(* CODESYS project CtaSysIO_1.0.0.1.library
   DocFormat: reStructuredText
   DefaultNamespace: CtaSysIO
   Version: 1.0.0.1
   Placeholder: CtaSysIO
   Company: CTA
   Description: Io System Library der CTA
   CompiledLibraryCompatibilityVersion: CODESYS V3.5 SP16 Patch 3
   LanguageModelAttribute: qualified-access-only
   Title: CtaSysIO
   Author: SIS

Project tree, tasks and I/O mapping:
  libraries: WagoSysDynamicIoMapping, 1.0.4.0 (WAGO); Standard, 3.5.18.0 (System); VisuDialogs, * (System); CtaSysConfig, 1.0.0.2 (CTA); CtaVisSymbols, 1.0.0.0 (CTA); VisuSymbols, 4.5.0.0 (System); CtaAppReport, 1.0.0.2 (CTA); CtaAppBmk, 1.0.0.0 (CTA); CtaAppInfluxLog, 1.0.0.1 (CTA); SysCom, 3.5.17.0 (System); CtaSysIO, 1.0.0.1 (CTA); CtaVisHelp, 1.0.0.0 (CTA); WagoSysVisuBACnet, 2.0.0.0 (WAGO); WagoVisuIcons, 1.1.0.5 (WAGO); WagoVisuIconsMaterialDesign, 1.0.0.0 (WAGO)
  40 Visualizations/
    AI/
      visualisation SimAI_Temp
      visualisation SimAI
      visualisation SimAI_Temp_Querry
    AO/
      visualisation SimAO_Temp
      visualisation SimAO
      visualisation SimAO_Temp_Querry
    DI/
      visualisation SimDI
      visualisation SimDI_Temp
      visualisation SimDI_Temp_Querry
    DO/
      visualisation SimDO_Temp
      visualisation SimDO
      visualisation SimDO_Temp_Querry
    Simulation/
      visualisation Simulation
      visualisation ModulInfos
      visualisation SimulationInfos
      visualisation DIA_IO_CONFIG
    Parameter/
      visualisation VIS_IO_PARAMETER_BASE
      Parameter_AI/
        visualisation VIS_PARAMETER_AI
        visualisation VIS_PARAMETER_TEMP_AI
      Parameter_DI/
        visualisation VIS_PARAMETER_DI
        visualisation VIS_PARAMETER_TEMP_DI
      Parameter_AO/
        visualisation VIS_PARAMETER_AO
        visualisation VIS_PARAMETER_TEMP_AO
      Parameter_DO/
        visualisation VIS_PARAMETER_DO
        visualisation VIS_PARAMETER_TEMP_DO
    PFC VISU/
      visualisation IO_ManagerBusInfo
      visualisation PFC_SLOT
      visualisation IO_Manager_Base
      visualisation IO_Manager_Sync
      visualisation IO_Manager_View
  30 Program Organization Units/
    fb/
      function block fbIO_Manager_Alt [ST]: proCycleStartDelayDone, metRequestIO_ITF, proAyIOs, proMaxIO, proErrNotEnoughIOs, proIoInitDone, proKbusErrHW, proKbusErrSW, proNeededMemSize, metRequestCOM_ITF, metModulConfigCheck
      HilfsFbs/
        function block fbIO [ST]: proSimVisu, proSlot, proChannelAdress, proPhysikalValueVisu, proOK, proKbusOk, proChannel, metCyclicKbus, proModuleType, proOkVisu, metConfig, P_scfbIO_fbxSimulationLock, P_scfbIO_Simulation, proIsHand, proAyPos, metTrendLog, proLogName, proIsBOOL_IO, proIoSim
        function block fbAI [ST]: proPhysikalValueVisu, proValue, metCyclicKbus, proAlUnterlauf, proPhysicalValue, proAlUeberlauf, proThisRef_AI, P_scfbAI_fbrMin, P_scfbAI_fbrMax, P_scfbAI_fbrMinPhysical, P_scfbAI_fbstPhysicalUnit, P_scfbAI_fbrPhysicalAlarm, P_scfbAI_fbrSimulationValue, P_scfbAI_fbrCorrectionValue, P_All_Init, metConfig, metTrendLog, proLogName, proIsBOOL_IO
        function block fbDO [ST]: proPhysikalValueVisu, proValue, metCyclicKbus, metConfig, proThisRef_DO, P_scfbDO_fbxInvert, P_scfbDO_fbxSimulationValue, P_All_Init, metTrendLog, proLogName, proIsBOOL_IO
        function block fbAO [ST]: proPhysikalValueVisu, metCyclicKbus, proValue, proPhysicalValue, metConfig, proThisRef_AO, P_scfbAO_fbrMin, P_scfbAO_fbrMax, P_scfbAO_fbrMinPhysical, P_scfbAO_fbrSimulationValue, P_All_Init, metTrendLog, proLogName, proIsBOOL_IO
        function block fbDI [ST]: proPhysikalValueVisu, metCyclicKbus, proValue, metConfig, proThisRef_DI, P_scfbDI_fbxInvert, P_scfbDI_fbxSimulationValue, P_All_Init, metTrendLog, proLogName, proIsBOOL_IO
      visuhilfe/
        function block fbPfcVisuHelp [ST]: metGetSlotIos, metNotShowChannel, proScrollBar, metCalcScrollBar, metCalcSlotFromScrollBar, getSizeOfFrame
      function block fbIO_Manager [ST]: proCycleStartDelayDone, metRequestIO_ITF, proAyIOs, proMaxIO, proErrNotEnoughIOs, proIoInitDone, proKbusErrHW, proKbusErrSW, proNeededMemSize, metRequestCOM_ITF, metModulConfigCheck, proSimOn, proAllowSim
    fc/
      Modul/
        function fcModuleType [ST]
      Adresse/
        function fcSlotAdress [ST]
      Skalierungen/
        function fcScaleIN4_20mA [ST]
        function fcScalePT1000 [ST]
        function fcSimValueScaler [ST]
        function fcScaleIN0_10V [ST]
        function fcScaleOut [ST]
      ITF_Prüfung/
        function fc_ITF_Evaluation [ST]
      Terminal Visu/
        function fcGetModulImage [ST]
        function fcSetModulImageForSimAndGetChanels [ST]
      ModulCheck/
        function fcCheckModul [ST]
    program IO [ST]
  00000000-0000-0000-0000-000000000000|D:\CoDeSys\LibrariesV3\trunk\Intern\CAA\CAA Template\3.4.0.0 draft\Placeholder.xml
  00000000-0000-0000-0000-000000000000|D:\CoDeSys\LibrariesV3\trunk\Intern\CAA\CAA Template\3.2.0.3 draft\Prefix.pdf
  00000000-0000-0000-0000-000000000000|D:\CoDeSys\LibrariesV3\trunk\Intern\CAA\CAA Template\3.5.2.0 draft\Placeholder.xml
  20 Structs/
    data type scChanelAdress
    data type enModuleType
    Parameter/
      data type scAI_Para
      data type scAO_Para
      data type scDI_Para
      data type scDO_Para
  50 Images/
    image pool IO_TERMINALS
  10 Documenation/
    global variables VersionHistory
    global variables readMe
  21 Interface/
    Visu/
      interface ITF_IO_Manager_Visu: proErrNotEnoughIOs, proNeededMemSize, proIoInitDone, proKbusErrSW, proKbusErrHW, proMaxIO, proAyIOs, proSimOn, proAllowSim
    IO/
      interface ITF_AI: proAlUnterlauf, proValue, proPhysicalValue, proAlUeberlauf, proThisRef_AI, P_scfbAI_fbrCorrectionValue, P_scfbAI_fbrMax, P_scfbAI_fbrMin, P_scfbAI_fbrMinPhysical, P_scfbAI_fbrPhysicalAlarm, P_scfbAI_fbrSimulationValue, P_scfbAI_fbstPhysicalUnit, P_All_Init
      interface ITF_AO: proPhysicalValue, proValue, proThisRef_AO, P_scfbAO_fbrMax, P_scfbAO_fbrMin, P_scfbAO_fbrMinPhysical, P_scfbAO_fbrSimulationValue, P_All_Init
      interface ITF_DI: proValue, proThisRef_DI, P_scfbDI_fbxInvert, P_scfbDI_fbxSimulationValue, P_All_Init
      interface ITF_DO: proValue, proThisRef_DO, P_scfbDO_fbxInvert, P_scfbDO_fbxSimulationValue, P_All_Init
      interface ITF_IO: proPhysikalValueVisu, proKbusOk, proOkVisu, proModuleType, proSimVisu, proOK, proSlot, proChannel, metCyclicKbus, proChannelAdress, P_scfbIO_fbxSimulationLock, P_scfbIO_Simulation, proIsHand, proLogName, proIsBOOL_IO, proIoSim
  11 Library Parameter/
    global variables Parameter
  12 Konstanten/
    global variables GlobalKonstant
  60 Textlisten/
    text list txtModulType
    text list txtWarning
    text list txtError
    text list txtPhysicalUnit
  13 Globale Variablen/
    global variables GVL_IO
    global variables GVL_IO_TERMINALS
  text list GlobalTextList
  5ce3da45-db07-42e7-a21c-a00fff4ed8f6|S:\_Temporär_SIS\CtaCodesysLibrary\01_Library\CtaSysIO\04_Image\0750_400.bmp
  5ce3da45-db07-42e7-a21c-a00fff4ed8f6|S:\_Temporär_SIS\CtaCodesysLibrary\01_Library\CtaSysIO\04_Image\0750_432.bmp
  5ce3da45-db07-42e7-a21c-a00fff4ed8f6|S:\_Temporär_SIS\CtaCodesysLibrary\01_Library\CtaSysIO\04_Image\0750_451.bmp
  5ce3da45-db07-42e7-a21c-a00fff4ed8f6|S:\_Temporär_SIS\CtaCodesysLibrary\01_Library\CtaSysIO\04_Image\0750_455.bmp
  5ce3da45-db07-42e7-a21c-a00fff4ed8f6|S:\_Temporär_SIS\CtaCodesysLibrary\01_Library\CtaSysIO\04_Image\0750_459.bmp
  5ce3da45-db07-42e7-a21c-a00fff4ed8f6|S:\_Temporär_SIS\CtaCodesysLibrary\01_Library\CtaSysIO\04_Image\0750_466.bmp
  5ce3da45-db07-42e7-a21c-a00fff4ed8f6|S:\_Temporär_SIS\CtaCodesysLibrary\01_Library\CtaSysIO\04_Image\0750_515.bmp
  5ce3da45-db07-42e7-a21c-a00fff4ed8f6|S:\_Temporär_SIS\CtaCodesysLibrary\01_Library\CtaSysIO\04_Image\0750_597.bmp
  5ce3da45-db07-42e7-a21c-a00fff4ed8f6|S:\_Temporär_SIS\CtaCodesysLibrary\01_Library\CtaSysIO\04_Image\0750_600.bmp
  5ce3da45-db07-42e7-a21c-a00fff4ed8f6|S:\_Temporär_SIS\CtaCodesysLibrary\01_Library\CtaSysIO\04_Image\0750_652.bmp
  5ce3da45-db07-42e7-a21c-a00fff4ed8f6|S:\_Temporär_SIS\CtaCodesysLibrary\01_Library\CtaSysIO\04_Image\0750_1405.bmp
  5ce3da45-db07-42e7-a21c-a00fff4ed8f6|S:\_Temporär_SIS\CtaCodesysLibrary\01_Library\CtaSysIO\04_Image\0750_1415.bmp
  5ce3da45-db07-42e7-a21c-a00fff4ed8f6|S:\_Temporär_SIS\CtaCodesysLibrary\01_Library\CtaSysIO\04_Image\0750_1504.bmp
  5ce3da45-db07-42e7-a21c-a00fff4ed8f6|S:\_Temporär_SIS\CtaCodesysLibrary\01_Library\CtaSysIO\04_Image\0750_8212.bmp
  5ce3da45-db07-42e7-a21c-a00fff4ed8f6|S:\_Temporär_SIS\CtaCodesysLibrary\01_Library\CtaSysIO\04_Image\0750_BLANK.bmp
  5ce3da45-db07-42e7-a21c-a00fff4ed8f6|S:\_Temporär_SIS\CtaCodesysLibrary\01_Library\CtaSysIO\04_Image\0750_555.bmp
*)

// 20 Structs/scChanelAdress
TYPE scChanelAdress :
STRUCT	
	uiByteNr	: 	UINT;
	uiBitNR		:	USINT;	
END_STRUCT
END_TYPE

// 20 Structs/enModuleType
{attribute 'qualified_only'}
{attribute 'strict'}
{attribute 'to_string'}
TYPE enModuleType :
(
	Unknown 		:= 0,
	Digital_IN		:= 1,
	Digital_OUT		:= 2,	
	DC_0_10V_OUT	:= 3,
	DC_4_20mA_OUT	:= 4,
	DC_0_10V_IN		:= 5,
	DC_4_20mA_IN	:= 6,
	OHM				:= 7,
    RS485			:= 8,
	DC_0_20mA_OUT	:= 9
);
END_TYPE

// 20 Structs/Parameter/scAI_Para
TYPE scAI_Para :
	STRUCT
		xSimulationLock		:	BOOL;
		rMin				:	REAL;
		rMax				:	REAL;
		rMinPhysical		:	REAL;
		rPhysicalAlarm		:	REAL;
		rCorrectionValue	:	REAL;
		stPhysicalUnit		:	STRING(40);
	END_STRUCT
END_TYPE

// 20 Structs/Parameter/scAO_Para
TYPE scAO_Para :
	STRUCT
		xSimulationLock		:	BOOL;
		rMin				:	REAL;
		rMax				:	REAL;
		rMinPhysical		:	REAL;
	END_STRUCT
END_TYPE

// 20 Structs/Parameter/scDI_Para
TYPE scDI_Para :
	STRUCT
		xSimulationLock		:	BOOL;
		xInvert				:	BOOL;
	END_STRUCT
END_TYPE

// 20 Structs/Parameter/scDO_Para
TYPE scDO_Para :
	STRUCT
		xSimulationLock		:	BOOL;
		xInvert				:	BOOL;
	END_STRUCT
END_TYPE

// 10 Documenation/VersionHistory
(* 

.. image:: ../../Images/CTA_Logo.jpg
   :align: right
   :width: 15% 

**Vorlage**   


============ =========== =========== ============================================
**Date**     **Version** **Author**  **Change**
------------ ----------- ----------- --------------------------------------------
04.03.2021   0.0.0.0     SIS         Vorlage erstellt

============ =========== =========== ============================================


*)
VAR_GLOBAL
    stInfo : STRING:= '0.0.0.0, Vorlage, CTA';
END_VAR

// 10 Documenation/readMe
(*

**ReadMe**
 
|	**Empfehlung**
|
|	Dokumentrieren Sie die Library für eine nachhaltige Entwicklung
|     
| *Beispiel*
| 
| Dies ist die Vorlage Library der CTA. Erstellen Sie ihre Library anhand dieser Vorlage.
*)

VAR_GLOBAL
    xReadMeDone              :   BOOL;
END_VAR

// 13 Globale Variablen/GVL_IO
{attribute 'qualified_only'}
VAR_GLOBAL	
	fbIO_Manager : fbIO_Manager;
END_VAR

// 11 Library Parameter/Parameter
{attribute 'qualified_only'}
VAR_GLOBAL CONSTANT
	SPS_BMK_ID        		: STRING(20)   := 'SPS';
	MAX_NUM_OF_DI			: INT := 200;
	MAX_NUM_OF_DO			: INT := 200;
	MAX_NUM_OF_AI			: INT := 100;
	MAX_NUM_OF_AO			: INT := 100;	
	                		
	MAX_NUM_OF_IOS			: INT := MAX_NUM_OF_DI + MAX_NUM_OF_DO + MAX_NUM_OF_AI + MAX_NUM_OF_AO;
	
	MAX_NUM_OF_COMTYPES		: INT := 10;
END_VAR

// 12 Konstanten/GlobalKonstant
{attribute 'qualified_only'}
VAR_GLOBAL CONSTANT
    stWarningTextList   :   STRING  := 'CtaSysIO.txtWarning';
    stErrorTextList     :   STRING  := 'CtaSysIO.txtError';
	ayMin	: ARRAY [enModuleType.Unknown..enModuleType.DC_0_20mA_OUT] OF REAL := [3(0), 0.0, 4, 0, 4, -250, 2(0.0)];
	ayMax	: ARRAY [enModuleType.Unknown..enModuleType.DC_0_20mA_OUT] OF REAL := [0, 2(1), 10, 20, 10, 20, 850, 0.0, 20];
END_VAR

// 13 Globale Variablen/GVL_IO_TERMINALS
{attribute 'qualified_only'}
VAR_GLOBAL
	aystIoTerminalType		:	ARRAY[1..125] OF STRING;
END_VAR

// 21 Interface/IO/ITF_AI
INTERFACE ITF_AI EXTENDS ITF_IO

PROPERTY proAlUnterlauf : BOOL
GET
END_GET
END_PROPERTY

PROPERTY proValue : REAL
GET
END_GET
END_PROPERTY

PROPERTY proPhysicalValue : REAL
GET
END_GET
END_PROPERTY

PROPERTY proAlUeberlauf : BOOL
GET
END_GET
END_PROPERTY

PROPERTY proThisRef_AI : REFERENCE TO fbAI
GET
END_GET
END_PROPERTY

PROPERTY P_scfbAI_fbrCorrectionValue : CtaSysConfig.ITF_DATATYPE
GET
END_GET
END_PROPERTY

PROPERTY P_scfbAI_fbrMax : CtaSysConfig.ITF_DATATYPE
GET
END_GET
END_PROPERTY

PROPERTY P_scfbAI_fbrMin : CtaSysConfig.ITF_DATATYPE
GET
END_GET
END_PROPERTY

PROPERTY P_scfbAI_fbrMinPhysical : CtaSysConfig.ITF_DATATYPE
GET
END_GET
END_PROPERTY

PROPERTY P_scfbAI_fbrPhysicalAlarm : CtaSysConfig.ITF_DATATYPE
GET
END_GET
END_PROPERTY

PROPERTY P_scfbAI_fbrSimulationValue : CtaSysConfig.ITF_DATATYPE
GET
END_GET
END_PROPERTY

PROPERTY P_scfbAI_fbstPhysicalUnit : CtaSysConfig.ITF_DATATYPE
GET
END_GET
END_PROPERTY

PROPERTY P_All_Init : scAI_Para
SET
END_SET
END_PROPERTY

END_INTERFACE

// 21 Interface/IO/ITF_IO
INTERFACE ITF_IO EXTENDS __system.IQueryInterface

PROPERTY proPhysikalValueVisu : STRING(6)
GET
END_GET
END_PROPERTY

PROPERTY proKbusOk : BOOL
GET
END_GET
SET
END_SET
END_PROPERTY

PROPERTY proOkVisu : STRING
GET
END_GET
END_PROPERTY

PROPERTY proModuleType : enModuleType
SET
END_SET
GET
END_GET
END_PROPERTY

PROPERTY proSimVisu : STRING
GET
END_GET
END_PROPERTY

PROPERTY proOK : BOOL
GET
END_GET
END_PROPERTY

PROPERTY proSlot : USINT
SET
END_SET
GET
END_GET
END_PROPERTY

PROPERTY proChannel : UINT
GET
END_GET
SET
END_SET
END_PROPERTY

METHOD metCyclicKbus
VAR_INPUT
END_VAR
END_METHOD

PROPERTY proChannelAdress : scChanelAdress
SET
END_SET
END_PROPERTY

PROPERTY P_scfbIO_fbxSimulationLock : CtaSysConfig.ITF_DATATYPE
GET
END_GET
END_PROPERTY

PROPERTY P_scfbIO_Simulation : CtaSysConfig.ITF_DATATYPE
GET
END_GET
END_PROPERTY

PROPERTY proIsHand : BOOL
GET
END_GET
END_PROPERTY

PROPERTY proLogName : STRING(100)
GET
END_GET
END_PROPERTY

PROPERTY proIsBOOL_IO : BOOL
GET
END_GET
END_PROPERTY

PROPERTY proIoSim : BOOL
SET
END_SET
GET
END_GET
END_PROPERTY

END_INTERFACE

// 30 Program Organization Units/fb/HilfsFbs/fbAI
FUNCTION_BLOCK fbAI EXTENDS fbIO IMPLEMENTS ITF_AI

VAR
	(*Channel input*)
	wChannelIn			: 	WORD;	
	
	(*Value output*)
	rValue				: 	REAL;
	
	(*Calculation Vars*)
	rPhysicalValueSIM	:	REAL;	// Errechneter Wert V oder mA der Simulation
	rPhysicalValuePLC 	:	REAL;	// Errechneter Wert V oder mA des PGMs
	rUserScale			:	REAL;  	// Funktionsausgabe, Physikalisch oder Benutzerdefiniert skaliert	
	
	(*Alarm*)	
	xAlUeberlauf		:	BOOL;	// Alarm Überlauf
	xAlUnterlauf		:	BOOL;	// Alarm Unterlauf
	(* Trendlog *)
	fbTrendLogrValue	:	CtaAppInfluxLog.FB_LOG_NODE_REAL;		
	(*Parameter*)	
	fbrMin				:	CtaSysConfig.fbREAL;			
	fbrMax				:	CtaSysConfig.fbREAL;		
	fbrMinPhysical		:	CtaSysConfig.fbREAL;
	fbstPhysicalUnit	:	CtaSysConfig.fbSTRING40;			
	fbrPhysicalAlarm	:	CtaSysConfig.fbREAL;			
	fbrSimulationValue	:	CtaSysConfig.fbREAL;
	fbrCorrectionValue	:	CtaSysConfig.fbREAL;			
END_VAR

PROPERTY proPhysikalValueVisu : STRING(6)
GET
// Schreiben des physikalischen Wertes für Visualisierung
IF FIND(TO_STRING(proPhysicalValue),'.') <> 0 THEN
	proPhysikalValueVisu := LEFT(TO_STRING(proPhysicalValue),(FIND(TO_STRING(proPhysicalValue),'.')+1));	
ELSE
	proPhysikalValueVisu := TO_STRING(proPhysicalValue);
END_IF
END_GET
END_PROPERTY

PROPERTY proValue : REAL
GET
(*Wert mit Korrektur*)
proValue := rValue;
END_GET
END_PROPERTY

METHOD FINAL metCyclicKbus
VAR
	xTempOk	:	BOOL;
END_VAR
metConfig();

// Lesen des Wertes aus definiertem Eingang
IF usiSlot > 0 AND WagoSysDynamicIoMapping.DynIoManager.DynKbusIoManager.coModules.uiModuleCount >= usiSlot THEN
	wChannelIn := WagoSysDynamicIoMapping.DynIoManager.DynKbusIoManager.coModules.aIModules[usiSlot].GetProcessInWord(scAdressOfChanel.uiByteNr,oStatus => oStatus);
ELSE
	wChannelIn 	:= 0;
	xOK			:= FALSE;
END_IF

// Modultyp bestimmen für physikalische Einheit
CASE enTypeOfModul OF
	enModuleType.DC_0_10V_IN,enModuleType.DC_0_10V_OUT:
		fbrSimulationValue.metNewMinMax(0,10); 
	enModuleType.DC_0_20mA_OUT:
		fbrSimulationValue.metNewMinMax(0,20); 
	enModuleType.DC_4_20mA_IN,enModuleType.DC_4_20mA_OUT:
		fbrSimulationValue.metNewMinMax(4,20);
	enModuleType.OHM:
		fbrSimulationValue.metNewMinMax(-2000,8500);
END_CASE	

// Signalausgabe an PGM, bei aktiver Simulation = Simulationswert
IF NOT fbxSimulation.xValue OR fbxSimulationLock.xValue THEN
      // Skalierung 0-10 V
	IF enTypeOfModul = enModuleType.DC_0_10V_IN THEN
		
		rUserScale := fcScaleIN0_10V(	wChanelInput 	:= 	wChannelIn,
										rMin 			:= 	fbrMin.rValue,
										rMax 			:= 	fbrMax.rValue,
										rMinPysical 	:=	fbrMinPhysical.rValue,
										rPysicalAlarm	:=	fbrPhysicalAlarm.rValue,									
										xOk				:= 	xOK,
										rV 				 => rPhysicalValuePLC,
										xAlUeberlauf 	 => xAlUeberlauf,
										xAlUnterlauf 	 => xAlUnterlauf);
										
	// Skalierung 4-20 mA	
	ELSIF enTypeOfModul = enModuleType.DC_4_20mA_IN THEN
	
		rUserScale := fcScaleIN4_20mA(	wChanelInput 	:= 	wChannelIn,
										rMin			:= 	fbrMin.rValue,
										rMax 			:= 	fbrMax.rValue,
										rmA 			 => rPhysicalValuePLC,
										xOK 			 => xOK,
										xAlUeberlauf 	 => xAlUeberlauf,
										xAlUnterlauf 	 => xAlUnterlauf);	

	// Skalierung ohm	
	ELSIF enTypeOfModul = enModuleType.ohm THEN
		
		rUserScale := fcScalePT1000(	wChanelInput	:=	wChannelIn,
										xOK 			 => xOK,
										xAlUeberlauf 	 => xAlUeberlauf,
										xAlUnterlauf 	 => xAlUnterlauf);
										
		rPhysicalValuePLC := rUserScale;

	END_IF
	
	// Übergabe des skalierten Eingangssignals
	rValue						:= rUserScale  + fbrCorrectionValue.rValue;
	fbrSimulationValue.metNewValueNoSave(proPhysicalValue);      
ELSE
	IF enTypeOfModul = enModuleType.ohm THEN
		rValue              := fbrSimulationValue.rValue;
		rPhysicalValueSIM   := fbrSimulationValue.rValue;    
	ELSE	
		// Skalierung des Simulationswertes
		rValue := fcSimValueScaler(	rSimulationValue 	:=	fbrSimulationValue.rValue,
									enIOModulType		:=	enTypeOfModul,
									rMin 				:= 	fbrMin.rValue,
									rMinPysical			:=	fbrMinPhysical.rValue,
									rMax				:=	fbrMax.rValue,
									rPysicalAlarm 		:=	fbrPhysicalAlarm.rValue,
									xOk 				:= 	xOK,
									xAlUnterlauf 		 => xAlUnterlauf);
		rPhysicalValueSIM := fbrSimulationValue.rValue;
	END_IF
END_IF

(* TREND *)
metTrendLog();
END_METHOD

PROPERTY proAlUnterlauf : BOOL
GET
proAlUnterlauf := xAlUnterlauf;
END_GET
END_PROPERTY

PROPERTY proPhysicalValue : REAL
GET
// Ausgabe Simulationswert bei aktiver Simulation
IF fbxSimulation.proValue THEN
	proPhysicalValue := rPhysicalValueSIM;
ELSE
	proPhysicalValue := rPhysicalValuePLC;
END_IF
END_GET
END_PROPERTY

PROPERTY proAlUeberlauf : BOOL
GET
proAlUeberlauf := xAlUeberlauf;
END_GET
END_PROPERTY

PROPERTY proThisRef_AI : REFERENCE TO fbAI
GET
proThisRef_AI REF= THIS^;
END_GET
END_PROPERTY

PROPERTY P_scfbAI_fbrMin : CtaSysConfig.ITF_DATATYPE
GET
P_scfbAI_fbrMin := fbrMin;
END_GET
END_PROPERTY

PROPERTY P_scfbAI_fbrMax : CtaSysConfig.ITF_DATATYPE
GET
P_scfbAI_fbrMax := fbrMax;
END_GET
END_PROPERTY

PROPERTY P_scfbAI_fbrMinPhysical : CtaSysConfig.ITF_DATATYPE
GET
P_scfbAI_fbrMinPhysical:= fbrMinPhysical;
END_GET
END_PROPERTY

PROPERTY P_scfbAI_fbstPhysicalUnit : CtaSysConfig.ITF_DATATYPE
GET
P_scfbAI_fbstPhysicalUnit := fbstPhysicalUnit;
END_GET
END_PROPERTY

PROPERTY P_scfbAI_fbrPhysicalAlarm : CtaSysConfig.ITF_DATATYPE
GET
P_scfbAI_fbrPhysicalAlarm := fbrPhysicalAlarm;
END_GET
END_PROPERTY

PROPERTY P_scfbAI_fbrSimulationValue : CtaSysConfig.ITF_DATATYPE
GET
P_scfbAI_fbrSimulationValue := fbrSimulationValue;
END_GET
END_PROPERTY

PROPERTY P_scfbAI_fbrCorrectionValue : CtaSysConfig.ITF_DATATYPE
GET
P_scfbAI_fbrCorrectionValue := fbrCorrectionValue;
END_GET
END_PROPERTY

PROPERTY P_All_Init : scAI_Para
SET
fbxSimulationLock._WertInit 	:= P_All_Init.xSimulationLock;
fbrMin._WertInit				:= P_All_Init.rMin;
fbrMax._WertInit				:= P_All_Init.rMax;
fbrMinPhysical._WertInit		:= P_All_Init.rMinPhysical;
fbrPhysicalAlarm._WertInit		:= P_All_Init.rPhysicalAlarm;
fbrCorrectionValue._WertInit	:= P_All_Init.rCorrectionValue;
fbstPhysicalUnit._WertInit		:= P_All_Init.stPhysicalUnit;
END_SET
END_PROPERTY

METHOD metConfig
VAR_INPUT
END_VAR
fbConfigFile();

fbxSimulation 					(_usiParaNr := 1, itfConfigFb := fbConfigFile);
fbxSimulationLock				(_usiParaNr := 2, itfConfigFb := fbConfigFile);
fbrMin							(_usiParaNr := 3, itfConfigFb := fbConfigFile);
fbrMax							(_usiParaNr := 4, itfConfigFb := fbConfigFile);
fbrMinPhysical					(_usiParaNr := 5, itfConfigFb := fbConfigFile);
fbrPhysicalAlarm				(_usiParaNr := 6, itfConfigFb := fbConfigFile);
fbrSimulationValue				(_usiParaNr := 7, itfConfigFb := fbConfigFile);
fbrCorrectionValue				(_usiParaNr := 8, itfConfigFb := fbConfigFile);
fbstPhysicalUnit				(_usiParaNr := 9, itfConfigFb := fbConfigFile);
END_METHOD

METHOD metTrendLog
IF NOT fbTrendLogrValue.ENABLE THEN
	fbTrendLogrValue.ENABLE	 := TRUE;
	fbTrendLogrValue.KEY	 := CONCAT('SLOT_',CONCAT(TO_STRING(usiSlot),CONCAT('_AI_',TO_STRING(uiChanel))));
END_IF;
fbTrendLogrValue.SET_VALUE	 := SEL(proIsHand,rPhysicalValuePLC,rPhysicalValueSIM);
END_METHOD

PROPERTY proLogName : STRING(100)
GET
proLogName := CONCAT('SLOT_',CONCAT(TO_STRING(usiSlot),CONCAT('_AI_',TO_STRING(uiChanel))));
END_GET
END_PROPERTY

PROPERTY proIsBOOL_IO : BOOL
GET
proIsBOOL_IO := FALSE;
END_GET
END_PROPERTY

END_FUNCTION_BLOCK

// 30 Program Organization Units/fb/HilfsFbs/fbIO
FUNCTION_BLOCK fbIO IMPLEMENTS ITF_IO
VAR_INPUT
END_VAR
VAR_OUTPUT
END_VAR
VAR	
	iAyPos				:	INT;
	xOK					: 	BOOL;
	xKbusOk				:	BOOL;
	xIoSim				:	BOOL;
	usiSlot				:	USINT;
	uiChanel			:	UINT;
	enTypeOfModul		:	enModuleType;
	scAdressOfChanel	: 	scChanelAdress;
	oStatus				: 	WagoSysErrorBase.FbResult;	
	
	(*Parameter*)
	fbConfigFile		: 	CtaSysConfig.fbConfigFile;

	fbxSimulation		:	CtaSysConfig.fbBOOL;
	fbxSimulationLock	:	CtaSysConfig.fbBOOL;	

END_VAR

PROPERTY proSimVisu : STRING
GET
// Simbolausgabe für Visu bei aktiver Simulations- Sperre
IF fbxSimulationLock.proValue THEN	
	proSimVisu := 'CtaVisSymbols.ImagePool.lock_closed_black';	
ELSE	
	IF fbxSimulation.proValue THEN
		proSimVisu := 'CtaVisSymbols.ImagePool.front_hand_Yellow';
	ELSE
		proSimVisu := '';
	END_IF	
END_IF
END_GET
END_PROPERTY

PROPERTY proSlot : USINT
SET
usislot := proSlot;
END_SET
GET
proSlot := usislot;
END_GET
END_PROPERTY

PROPERTY proChannelAdress : scChanelAdress
SET
scAdressOfChanel := proChannelAdress;
END_SET
END_PROPERTY

PROPERTY proPhysikalValueVisu : STRING(6)
GET
END_GET
SET
END_SET
END_PROPERTY

PROPERTY proOK : BOOL
GET
// Setzen des Modul OKs 
IF xOK AND xKbusOk THEN
	proOK := TRUE;
ELSIF xIoSim THEN
	proOK := TRUE;
ELSE
	proOK := FALSE;
END_IF
END_GET
END_PROPERTY

PROPERTY proKbusOk : BOOL
GET
 proKbusOk := xKbusOk;
END_GET
SET
xKbusOk := proKbusOk;
END_SET
END_PROPERTY

PROPERTY proChannel : UINT
SET
uiChanel := proChannel;
END_SET
GET
proChannel := uiChanel;
END_GET
END_PROPERTY

METHOD metCyclicKbus
END_METHOD

PROPERTY proModuleType : enModuleType
GET
proModuleType := enTypeOfModul;
END_GET
SET
enTypeOfModul := proModuleType;
END_SET
END_PROPERTY

PROPERTY proOkVisu : STRING
GET
// Definition des anzuzeigenden Bildes für Visu
IF xOK AND xKbusOk THEN
	proOkVisu := 'CtaVisSymbols.ImagePool.check_green';
ELSIF xIoSim THEN
	proOkVisu := 'CtaVisSymbols.ImagePool.front_hand_Yellow';
ELSE
	proOkVisu := 'CtaVisSymbols.ImagePool.CtaError';
END_IF
END_GET
END_PROPERTY

METHOD metConfig
VAR_INPUT
END_VAR
fbConfigFile();

fbxSimulation 					(_usiParaNr := 1, itfConfigFb := fbConfigFile,);
fbxSimulationLock				(_usiParaNr := 2, itfConfigFb := fbConfigFile,);
END_METHOD

PROPERTY P_scfbIO_fbxSimulationLock : CtaSysConfig.ITF_DATATYPE
GET
P_scfbIO_fbxSimulationLock := fbxSimulationLock;
END_GET
END_PROPERTY

PROPERTY P_scfbIO_Simulation : CtaSysConfig.ITF_DATATYPE
GET
P_scfbIO_Simulation := fbxSimulation;
END_GET
END_PROPERTY

PROPERTY proIsHand : BOOL
GET
proIsHand := NOT fbxSimulationLock.xValue AND fbxSimulation.xValue;
END_GET
END_PROPERTY

PROPERTY proAyPos : UINT
SET
iAyPos := TO_INT(proAyPos);
END_SET
GET
proAyPos := TO_UINT(iAyPos);
END_GET
END_PROPERTY

METHOD metTrendLog
END_METHOD

PROPERTY proLogName : STRING(100)
GET
proLogName := '';
END_GET
END_PROPERTY

PROPERTY proIsBOOL_IO : BOOL
GET
proIsBOOL_IO := FALSE;
END_GET
END_PROPERTY

PROPERTY proIoSim : BOOL
SET
xIoSim := proIoSim;
END_SET
GET
proiosim := xIoSim;
END_GET
END_PROPERTY

END_FUNCTION_BLOCK

// 30 Program Organization Units/fc/Skalierungen/fcScaleIN0_10V
FUNCTION fcScaleIN0_10V : Real
VAR_INPUT
	wChanelInput	: WORD;
	
	// Values for scaling
	rMin			:	REAL;
	rMinPysical		:	REAL;
	rMax			:	REAL;	
	rPysicalAlarm	:	REAL;	
END_VAR
VAR
	iChanelInput	: INT;
END_VAR
VAR_OUTPUT
	rV				: REAL;
	xAlUeberlauf	: BOOL;
	xAlUnterlauf	: BOOL;
END_VAR
VAR_IN_OUT
	xOk				: 	BOOL;
END_VAR

IF wChanelInput.0 = FALSE AND wChanelInput.1 = FALSE THEN
	// Für 12Bit Messwertausgabe die 3 Status Bit weglassen. Bit 16 kann vernachläsigt werden, da es immer 0 ist.
	iChanelInput 			:= WORD_TO_INT(SHR(wChanelInput,3)); 			// Prozesswert des AD Wandlers in INT										
	rV	   					:= INT_TO_REAL(iChanelInput) /(4095.0/10.0);	// Skalierung des Messwertes auf 0-10V
	// Prüfen ob die Skalierung machbar ist
	IF rMax - rMin <> 0 THEN	
		// Skalieren des Messwertes
		fcScaleIN0_10V		:= (INT_TO_REAL(iChanelInput)-(rMinPysical*4095/10)) * ((  rMax - rMin)/(4095.0-(rMinPysical*4095/10))) + rMin;  
	ELSE
		fcScaleIN0_10V		:= rV;	
	END_IF;
	// Schaltung: Messwert in Range
    IF rV >= rMinPysical THEN
        xOK             	:= TRUE;
	ELSIF rV < rMinPysical AND rV > (rMinPysical-((rMinPysical - rPysicalAlarm)/3)) THEN
		fcScaleIN0_10V  	:= rMin;
	ELSIF rV <= (rMinPysical-((rMinPysical - rPysicalAlarm)/3)) THEN
		xOK             	:= FALSE;    
        fcScaleIN0_10V  	:= rMin;
    END_IF;
	    
	// Störung: Sensorleitung ist Unterbrochen		
	IF rV < rPysicalAlarm THEN
        fcScaleIN0_10V   	:= 0; 	
        xAlUnterlauf     	:= TRUE;
        xOK              	:= FALSE;
	END_IF;
// Störung: Sensorleitung ist Unterbrochen	
ELSIF wChanelInput.0 = TRUE	AND wChanelInput.1 = TRUE THEN
	xAlUnterlauf			:= TRUE;
    fcScaleIN0_10V			:= -3.402823E+38;
	xOK						:= FALSE;
// Störung: Sensorleitung hat Überlauf	
ELSIF wChanelInput.0 = TRUE AND wChanelInput.1 = FALSE THEN
	xAlUeberlauf            := TRUE;
   	fcScaleIN0_10V          := 3.402823E+38;
	xOK						:= FALSE;
END_IF

END_FUNCTION

// 30 Program Organization Units/fc/Skalierungen/fcScaleIN4_20mA
FUNCTION fcScaleIN4_20mA : REAL
VAR_INPUT
	wChanelInput	: WORD;
	rMin        	: REAL;
    rMax        	: REAL;  
END_VAR	
VAR
	iChanelInput	: INT;	
END_VAR
VAR_OUTPUT
	rmA				: REAL;
	xOK				: BOOL;
	xAlUeberlauf	: BOOL;
	xAlUnterlauf	: BOOL;
END_VAR

//  Prüfen der Error Bit 0 & Bit 1 
IF wChanelInput.0 = FALSE AND wChanelInput.1 = FALSE THEN
	// Für 12Bit Messwertausgabe die 3 Status Bit weglassen. Bit 16 kann vernachläsigt werden, da es immer 0 ist.
	iChanelInput 			:= WORD_TO_INT(SHR(wChanelInput,3)); 					// Prozesswert des AD Wandlers in INt										
	rmA	   					:= INT_TO_REAL(iChanelInput) /(4095.0/16.0) + 4.0;		// Skalierung des Messwertes auf 4-20Ma
	// Prüfen ob die Skalierung machbar ist
	IF rMax - rMin <> 0 THEN	
		// Skalieren des Messwertes
		fcScaleIN4_20mA		:= INT_TO_REAL(iChanelInput)/(4095.0/(rMax - rMin)) + rMin; 
	ELSE
		fcScaleIN4_20mA		:= rmA;	 
	END_IF;
    xOK                 	:= TRUE;
// Störung: Sensorleitung ist Unterbrochen	
ELSIF wChanelInput.0 = TRUE AND wChanelInput.1 = TRUE THEN 
    xAlUnterlauf        	:= TRUE;
    fcScaleIN4_20mA     	:= 1.0E-44;
    xOK                 	:= FALSE;
// Störung: Sensorleitung hat Überlauf	
ELSIF wChanelInput.0 = TRUE AND wChanelInput.1 = FALSE THEN
    xAlUeberlauf        	:= TRUE;
    fcScaleIN4_20mA     	:= 3.402823E+38;
    xOK						:= FALSE;
END_IF;

END_FUNCTION

// 30 Program Organization Units/fc/Skalierungen/fcScalePT1000
FUNCTION fcScalePT1000 : REAL
VAR_INPUT
	wChanelInput	: WORD;
END_VAR
VAR
	iChanelInput	: INT;	
END_VAR

VAR_OUTPUT
	xOK				: BOOL;
	xAlUeberlauf	: BOOL;
	xAlUnterlauf	: BOOL;
END_VAR

// Prüfen ob der Wert gültig ist
iChanelInput := TO_INT(wChanelInput);
IF iChanelInput > -2000 AND iChanelInput < 8500 THEN   
	// Temperaturausgabe
	fcScalePT1000		:= INT_TO_REAL(iChanelInput)/10.0;
    xOK                 := TRUE;
// Störung: Sensorleitung ist Unterbrochen	
ELSIF iChanelInput >= 8500 THEN
    xAlUnterlauf        := TRUE;
    fcScalePT1000       := 1.0E-44;    
    xOK                 := FALSE;
// Störung: Sensorleitung hat Kurzschluss	
ELSIF iChanelInput <= -2000  THEN 
    xAlUeberlauf        := TRUE;
    fcScalePT1000       := 3.402823E+38;   
    xOK                 := FALSE;   
END_IF;

END_FUNCTION

// 30 Program Organization Units/fc/Skalierungen/fcSimValueScaler
FUNCTION fcSimValueScaler : REAL
VAR_INPUT
	rSimulationValue	: REAL;
	enIOModulType		: enModuleType;
	
	// Values for scaling
	rMin			:	REAL;
	rMinPysical		:	REAL;
	rMax			:	REAL;	
	rPysicalAlarm	:	REAL;	
END_VAR
VAR
	rMin_mA			:	REAL := 4;
	rMax_mA			:	REAL := 20;
	rMax_V			: 	REAL := 10;
	srSet			:	Standard.SR;
END_VAR
VAR_OUTPUT
	xAlUnterlauf	: 	BOOL;
END_VAR
VAR_IN_OUT
	xOk				: 	BOOL;
END_VAR

// 0 - 10 Volt
IF enIOModulType = enModuleType.DC_0_10V_IN OR enIOModulType = enModuleType.DC_0_10V_OUT THEN

	// Prüfen ob die Skalierung machbar ist
	IF rMax - rMin <> 0 THEN	
		// Skalieren des Messwertes
		fcSimValueScaler		:=  (rSimulationValue-(rMinPysical*rMax_V/10)) * ((  rMax - rMin)/(rMax_V-(rMinPysical*rMax_V/10))) + rMin;  
	ELSE
		fcSimValueScaler		:=  rSimulationValue;	
	END_IF;		
	
 	// Schaltung: Messwert in Range
    IF rSimulationValue >= rMinPysical THEN
		xOk := TRUE;		
	ELSIF rSimulationValue < rMinPysical AND rSimulationValue > (rMinPysical - ((rMinPysical - rPysicalAlarm)/3)) THEN
		fcSimValueScaler     	:=  rMin;
	ELSIF rSimulationValue <= (rMinPysical - ((rMinPysical - rPysicalAlarm)/3)) THEN
		xOk := FALSE;	 
        fcSimValueScaler     	:=  rMin;
	END_IF 
  
// Störung: Sensorleitung ist Unterbrochen		
	IF rSimulationValue < rPysicalAlarm THEN
        fcSimValueScaler    	:=  0; 	
        xAlUnterlauf        	:=  TRUE;
        xOk              		:=  FALSE;
	END_IF;
	
// 4 - 20 mA
ELSIF enIOModulType = enModuleType.DC_4_20mA_IN OR enIOModulType = enModuleType.DC_4_20mA_OUT THEN
	// Prüfen ob die Skalierung machbar ist
	IF rMax - rMin <> 0 THEN	
		// Skalieren des Messwertes
		fcSimValueScaler		:=  (rSimulationValue-(rMin_mA*rMax_mA/20)) * ((  rMax - rMin)/(rMax_mA-(rMin_mA*rMax_mA/20))) + rMin;  
		xOk 					:=  TRUE;
	ELSE
		fcSimValueScaler		:=  rSimulationValue;	
		xOk 					:=  TRUE; 
	END_IF;
// 4 - 20 mA
ELSIF enIOModulType = enModuleType.DC_0_20mA_OUT OR enIOModulType = enModuleType.DC_0_20mA_OUT THEN
	// Prüfen ob die Skalierung machbar ist
	IF rMax - rMin <> 0 THEN	
		// Skalieren des Messwertes
		fcSimValueScaler		:=  (rSimulationValue-(0*rMax_mA/20)) * ((  rMax - rMin)/(rMax_mA-(0*rMax_mA/20))) + rMin;  
		xOk 					:=  TRUE;
	ELSE
		fcSimValueScaler		:=  rSimulationValue;	
		xOk 					:=  TRUE; 
	END_IF;	
// ohm 
ELSIF enIOModulType = enModuleType.ohm THEN
	fcSimValueScaler := rSimulationValue; 
	xOk 					:=  TRUE;
END_IF

END_FUNCTION

// 21 Interface/IO/ITF_AO
INTERFACE ITF_AO EXTENDS ITF_IO

PROPERTY proPhysicalValue : REAL
GET
END_GET
END_PROPERTY

PROPERTY proValue : REAL
SET
END_SET
GET
END_GET
END_PROPERTY

PROPERTY proThisRef_AO : REFERENCE TO fbAO
GET
END_GET
END_PROPERTY

PROPERTY P_scfbAO_fbrMax : CtaSysConfig.ITF_DATATYPE
GET
END_GET
END_PROPERTY

PROPERTY P_scfbAO_fbrMin : CtaSysConfig.ITF_DATATYPE
GET
END_GET
END_PROPERTY

PROPERTY P_scfbAO_fbrMinPhysical : CtaSysConfig.ITF_DATATYPE
GET
END_GET
END_PROPERTY

PROPERTY P_scfbAO_fbrSimulationValue : CtaSysConfig.ITF_DATATYPE
GET
END_GET
END_PROPERTY

PROPERTY P_All_Init : scAO_Para
SET
END_SET
END_PROPERTY

END_INTERFACE

// 30 Program Organization Units/fb/HilfsFbs/fbAO
FUNCTION_BLOCK fbAO EXTENDS fbIO IMPLEMENTS ITF_AO

VAR
	// Übergabewert des PGMs
	rValueIn: REAL;
		
	// Calculated value
	rPhysicalValue	: 	REAL;	// Errechneter phyikalischer Wert
	
	// Transfer variable
	wValueOut		:	WORD;	// Übergabevariable
	
	// Channel output
	wChannelOut		: 	WORD;	
	(* Trendlog *)
	fbTrendLogrValue	:	CtaAppInfluxLog.FB_LOG_NODE_REAL;	
	(*Parameter*)
	fbrMin				: ctasysConfig.fbreAL;
	fbrMax				: ctasysConfig.fbreAL;
	fbrMinPhysical		: ctasysConfig.fbreAL;
	fbrSimulationValue	: ctasysConfig.fbreAL;	
END_VAR

PROPERTY proPhysikalValueVisu : String(6)
GET
// Schreiben des physikalischen Wertes für Visualisierung
IF proPhysicalValue >= 10 THEN
	proPhysikalValueVisu := LEFT(TO_STRING(proPhysicalValue),4);
ELSE
	proPhysikalValueVisu := LEFT(TO_STRING(proPhysicalValue),3);
END_IF
END_GET
END_PROPERTY

METHOD FINAL metCyclicKbus
metConfig();

// Bei aktiver Simulation wird Simulationswert ausgegeben
IF fbxSimulation.xValue AND NOT fbxSimulationLock.xValue THEN
	// Skalierung und Übergabe des Simulationswertes 0 - 10 V
	IF enTypeOfModul = enModuleType.DC_0_10V_OUT THEN
		wValueOut := fcScaleOut(	rValueIn 			:= 	fbrSimulationValue.rValue,
									rMinPhysicalValue 	:= 	fbrMinPhysical.rValue,
									rMin 				:= 	0,
									rMax 				:= 	10,
									enTypeofModule 		:= 	enTypeOfModul,
									rPhysicalValue 		 =>	rPhysicalValue);
		fbrSimulationValue.metNewMinMax(0,10);  
	
	// Skalierung und Übergabe des Simulationswertes 4 - 20 mA	
	ELSIF  enTypeOfModul = enModuleType.DC_4_20mA_OUT THEN
		wValueOut := fcScaleOut(	rValueIn 			:=	fbrSimulationValue.rValue,
									rMinPhysicalValue	:=	fbrMinPhysical.rValue,
									rMin 				:= 	4,
									rMax 				:= 	20,
									enTypeofModule 		:= 	enTypeOfModul,
									rPhysicalValue 		 => rPhysicalValue);
		fbrSimulationValue.metNewMinMax(4,20);  								
	// Skalierung und Übergabe des Simulationswertes 0 - 20 mA	
	ELSIF  enTypeOfModul = enModuleType.DC_4_20mA_OUT THEN
		wValueOut := fcScaleOut(	rValueIn 			:=	fbrSimulationValue.rValue,
									rMinPhysicalValue	:=	fbrMinPhysical.rValue,
									rMin 				:= 	0,
									rMax 				:= 	20,
									enTypeofModule 		:= 	enTypeOfModul,
									rPhysicalValue 		 => rPhysicalValue); 									
	END_IF	
ELSE
	CASE enTypeOfModul OF
		enModuleType.DC_0_10V_IN,enModuleType.DC_0_10V_OUT:
			fbrSimulationValue.metNewMinMax(0,10); 
		enModuleType.DC_0_20mA_OUT:
			fbrSimulationValue.metNewMinMax(0,20); 
		enModuleType.DC_4_20mA_IN,enModuleType.DC_4_20mA_OUT:
			fbrSimulationValue.metNewMinMax(4,20);
		enModuleType.OHM:
			fbrSimulationValue.metNewMinMax(-2000,8500);
	END_CASE	
	// Skalierung und Übergabe des PGM- Wertes
	wValueOut := fcScaleOut(	rValueIn 			:=	rValueIn,
								rMinPhysicalValue	:= 	fbrMinPhysical.rValue,
								rMin				:= 	fbrMin.rValue,
								rMax				:= 	fbrMax.rValue,
								enTypeofModule		:= 	enTypeOfModul,
								rPhysicalValue 		 => rPhysicalValue);
								
	fbrSimulationValue.metNewValueNoSave(rPhysicalValue);
END_IF

wChannelOut := wValueOut;

// Write value on defined AO
IF usiSlot > 0 AND WagoSysDynamicIoMapping.DynIoManager.DynKbusIoManager.coModules.uiModuleCount >= usiSlot THEN
	WagoSysDynamicIoMapping.DynIoManager.DynKbusIoManager.coModules.aIModules[usiSlot].SetProcessOutWord(scAdressOfChanel.uiByteNr,wChannelOut,oStatus => oStatus);
	xOK := TRUE;
ELSE
	xOK := FALSE;
END_IF
	
(* TREND *)
metTrendLog();
END_METHOD

PROPERTY proValue : REAL
GET
proValue := rPhysicalValue;
END_GET
SET
rValueIn := proValue;
END_SET
END_PROPERTY

PROPERTY proPhysicalValue : REAL
GET
proPhysicalValue := rPhysicalValue;
END_GET
END_PROPERTY

METHOD metConfig
VAR_INPUT
END_VAR
fbConfigFile();

fbxSimulation 					(_usiParaNr := 1, itfConfigFb := fbConfigFile);
fbxSimulationLock				(_usiParaNr := 2, itfConfigFb := fbConfigFile);
fbrMin							(_usiParaNr := 3, itfConfigFb := fbConfigFile);
fbrMax							(_usiParaNr := 4, itfConfigFb := fbConfigFile);
fbrMinPhysical					(_usiParaNr := 5, itfConfigFb := fbConfigFile);
fbrSimulationValue				(_usiParaNr := 7, itfConfigFb := fbConfigFile);
END_METHOD

PROPERTY proThisRef_AO : REFERENCE TO fbAO
GET
proThisRef_AO REF= THIS^;
END_GET
END_PROPERTY

PROPERTY P_scfbAO_fbrMin : CtaSysConfig.ITF_DATATYPE
GET
P_scfbAO_fbrMin := fbrMin;
END_GET
END_PROPERTY

PROPERTY P_scfbAO_fbrMax : CtaSysConfig.ITF_DATATYPE
GET
P_scfbAO_fbrMax := fbrMax;
END_GET
END_PROPERTY

PROPERTY P_scfbAO_fbrMinPhysical : CtaSysConfig.ITF_DATATYPE
GET
P_scfbAO_fbrMinPhysical := fbrMinPhysical;
END_GET
END_PROPERTY

PROPERTY P_scfbAO_fbrSimulationValue : CtaSysConfig.ITF_DATATYPE
GET
P_scfbAO_fbrSimulationValue := fbrSimulationValue;
END_GET
END_PROPERTY

PROPERTY P_All_Init : scAO_Para
SET
fbxSimulationLock._WertInit := P_All_Init.xSimulationLock;
fbrMin._WertInit			:= P_All_Init.rMin;
fbrMax._WertInit			:= P_All_Init.rMax;
fbrMinPhysical._WertInit	:= P_All_Init.rMinPhysical;
END_SET
END_PROPERTY

METHOD metTrendLog
IF NOT fbTrendLogrValue.ENABLE THEN
	fbTrendLogrValue.ENABLE := TRUE;
	fbTrendLogrValue.KEY	 := CONCAT('SLOT_',CONCAT(TO_STRING(usiSlot),CONCAT('_AO_',TO_STRING(uiChanel))));
END_IF;
fbTrendLogrValue.SET_VALUE	 := rPhysicalValue;
END_METHOD

PROPERTY proLogName : STRING(100)
GET
proLogName := CONCAT('SLOT_',CONCAT(TO_STRING(usiSlot),CONCAT('_AO_',TO_STRING(uiChanel))));
END_GET
END_PROPERTY

PROPERTY proIsBOOL_IO : BOOL
GET
proIsBOOL_IO := FALSE;
END_GET
END_PROPERTY

END_FUNCTION_BLOCK

// 30 Program Organization Units/fc/Skalierungen/fcScaleOut
FUNCTION fcScaleOut : WORD
VAR_INPUT
	rValueIn			: REAL;
	rMinPhysicalValue	: REAL;
	rMin				: REAL;
	rMax				: REAL;
	enTypeofModule		: enModuleType;
END_VAR
VAR
	wMinCalcValue		: WORD;
	rPyhsicalMin		: REAL;
	rPysiclalMax		: REAL;
END_VAR
VAR_OUTPUT
	rPhysicalValue		: REAL;	
END_VAR

// Prüfen des Modultyps zur definition von Min / Max
IF enTypeofModule = enModuleType.DC_0_10V_OUT THEN	
	rPyhsicalMin		:= 0;
	rPysiclalMax		:= 10;	
ELSIF enTypeofModule = enModuleType.DC_4_20mA_OUT THEN
	rPyhsicalMin		:= 4;
	rPysiclalMax		:= 20;	
ELSIF enTypeofModule = enModuleType.DC_0_20mA_OUT THEN
	rPyhsicalMin		:= 0;
	rPysiclalMax		:= 20;		
END_IF

// Errechnung des minimalen Phyikalischen wertes
 wMinCalcValue   	:=  TO_WORD(TO_WORD(LIMIT(0,((LIMIT(rPyhsicalMin,rMinPhysicalValue,rPysiclalMax) - rPyhsicalMin)*((32767.0 - 0)/(rPysiclalMax-0)) + 0),32767)));
    
// Prüfen ob die Skalierung machbar ist
IF rMax - rMin <> 0 THEN	
    // Skalieren des Messwertes
   	fcScaleOut    		:=  TO_WORD(LIMIT(wMinCalcValue,(rValueIn - rMin)*((32767 - wMinCalcValue) / (rMax-rMin))+ wMinCalcValue,32767));
    rPhysicalValue    	:=  LIMIT(0,(TO_REAL(fcScaleOut) - 0)*((rPysiclalMax - rPyhsicalMin) / (32767-0))+ rPyhsicalMin,rPysiclalMax);    
ELSE
	// Ausgabe des minimalen Wertes falls Skallierung nicht möglich
    fcScaleOut    		:=  wMinCalcValue;	
    rPhysicalValue     	:=  LIMIT(rPyhsicalMin,rMinPhysicalValue,rPysiclalMax);
END_IF;

END_FUNCTION

// 21 Interface/IO/ITF_DI
INTERFACE ITF_DI EXTENDS ITF_IO

PROPERTY proValue : BOOL
GET
END_GET
END_PROPERTY

PROPERTY proThisRef_DI : REFERENCE TO fbDI
GET
END_GET
END_PROPERTY

PROPERTY P_scfbDI_fbxInvert : CtaSysConfig.ITF_DATATYPE
GET
END_GET
END_PROPERTY

PROPERTY P_scfbDI_fbxSimulationValue : CtaSysConfig.ITF_DATATYPE
GET
END_GET
END_PROPERTY

PROPERTY P_All_Init : scDI_Para
SET
END_SET
END_PROPERTY

END_INTERFACE

// 30 Program Organization Units/fb/HilfsFbs/fbDI
FUNCTION_BLOCK fbDI EXTENDS fbIO IMPLEMENTS ITF_DI

VAR
	// Channel input
	xChannelIn	:	BOOL;
	
	// Übergabe variablen
	xValue		:	BOOL;
	(* Trendlog *)
	fbTrendLogxValue				:	CtaAppInfluxLog.FB_LOG_NODE_BOOL;	
	(*Parameter*)
	fbxInvert			: ctasysConfig.fbBOOL;
	fbxSimulationValue	: ctasysConfig.fbBOOL;
END_VAR

PROPERTY proPhysikalValueVisu : String(6)
GET
// Schreiben des physikalischen Wertes für Visualisierung 
proPhysikalValueVisu := TO_STRING(proValue);
END_GET
END_PROPERTY

METHOD FINAL metCyclicKbus
metConfig();
// Read value from defined DI
IF usiSlot > 0 AND WagoSysDynamicIoMapping.DynIoManager.DynKbusIoManager.coModules.uiModuleCount >= usiSlot THEN
	xChannelIn := WagoSysDynamicIoMapping.DynIoManager.DynKbusIoManager.coModules.aIModules[usiSlot].GetProcessInBit(scAdressOfChanel.uiByteNr,scAdressOfChanel.uiBitNR,oStatus => oStatus);
	xOK := TRUE;
ELSE
	xOK := FALSE;
END_IF	
// Bei aktivierter Simulation wird der Simulationswert übertragen
IF fbxSimulation.xValue AND NOT fbxSimulationLock.xValue THEN
	xValue := fbxSimulationValue.xValue;
ELSE
	xValue := xChannelIn;
	fbxSimulationValue.metNewValueNoSave(xChannelIn);
END_IF
(* TREND *)
metTrendLog();
END_METHOD

PROPERTY proValue : BOOL
GET
// Invertierung des Wertes bei aktiver Invertierung
proValue := xValue XOR fbxInvert.proValue;
END_GET
END_PROPERTY

METHOD metConfig
VAR_INPUT
END_VAR
fbConfigFile();

fbxSimulation 					(_usiParaNr := 1, itfConfigFb := fbConfigFile);
fbxSimulationLock				(_usiParaNr := 2, itfConfigFb := fbConfigFile);
fbxInvert						(_usiParaNr := 3, itfConfigFb := fbConfigFile);
fbxSimulationValue				(_usiParaNr := 4, itfConfigFb := fbConfigFile);
END_METHOD

PROPERTY proThisRef_DI : REFERENCE TO fbDI
GET
proThisRef_DI REF= THIS^;
END_GET
END_PROPERTY

PROPERTY P_scfbDI_fbxInvert : CtaSysConfig.ITF_DATATYPE
GET
P_scfbDI_fbxInvert := fbxInvert;
END_GET
END_PROPERTY

PROPERTY P_scfbDI_fbxSimulationValue : CtaSysConfig.ITF_DATATYPE
GET
P_scfbDI_fbxSimulationValue := fbxSimulationValue;
END_GET
END_PROPERTY

PROPERTY P_All_Init : scDI_Para
SET
fbxSimulationLock._WertInit := P_All_Init.xSimulationLock;
fbxInvert._WertInit 		:= P_All_Init.xInvert;
END_SET
END_PROPERTY

METHOD metTrendLog
IF NOT fbTrendLogxValue.ENABLE THEN
	fbTrendLogxValue.ENABLE := TRUE;
	fbTrendLogxValue.KEY 	:= CONCAT('SLOT_',CONCAT(TO_STRING(usiSlot),CONCAT('_DI_',TO_STRING(uiChanel))));
END_IF;
fbTrendLogxValue.SET_VALUE	 := xValue;
END_METHOD

PROPERTY proLogName : STRING(100)
GET
proLogName := CONCAT('SLOT_',CONCAT(TO_STRING(usiSlot),CONCAT('_DI_',TO_STRING(uiChanel))));
END_GET
END_PROPERTY

PROPERTY proIsBOOL_IO : BOOL
GET
proIsBOOL_IO := TRUE;
END_GET
END_PROPERTY

END_FUNCTION_BLOCK

// 21 Interface/IO/ITF_DO
INTERFACE ITF_DO EXTENDS ITF_IO

PROPERTY proValue : BOOL
GET
END_GET
SET
END_SET
END_PROPERTY

PROPERTY proThisRef_DO : REFERENCE TO fbDO
GET
END_GET
END_PROPERTY

PROPERTY P_scfbDO_fbxInvert : CtaSysConfig.ITF_DATATYPE
GET
END_GET
END_PROPERTY

PROPERTY P_scfbDO_fbxSimulationValue : CtaSysConfig.ITF_DATATYPE
GET
END_GET
END_PROPERTY

PROPERTY P_All_Init : scDO_Para
SET
END_SET
END_PROPERTY

END_INTERFACE

// 30 Program Organization Units/fb/HilfsFbs/fbDO
FUNCTION_BLOCK fbDO EXTENDS fbIO IMPLEMENTS ITF_DO

VAR
	// Value in
	xValueIn	:	BOOL;
	
	// Transfer variable	
	xValue		:	BOOL;
		
	// Channel output
	xChannelOut	:	BOOL;
	(* Trendlog *)
	fbTrendLogxValue				:	CtaAppInfluxLog.FB_LOG_NODE_BOOL;
	(*Parameter*)
	fbxInvert						:	CtaSysConfig.fbBOOL;
	fbxSimulationValue				:	CtaSysConfig.fbBOOL;

END_VAR

PROPERTY proPhysikalValueVisu : String(6)
GET
// Schreiben des physikalischen Wertes für Visualisierung
proPhysikalValueVisu := TO_STRING(xChannelOut);
END_GET
END_PROPERTY

PROPERTY proValue : BOOL
GET
proValue := xValue;
END_GET
SET
xValueIn := proValue;
END_SET
END_PROPERTY

METHOD FINAL metCyclicKbus
metConfig();
// Bei aktiver Simulation wird Simulationswert dem Ausgang übergeben
IF fbxSimulation.xValue AND NOT fbxSimulationLock.xValue THEN
	xValue 	:= fbxSimulationValue.xValue;
ELSE
	xValue	:= xValueIn;
	fbxSimulationValue.metNewValueNoSave(xValueIn);
END_IF

IF NOT proKbusOk AND NOT xIoSim THEN
	// Abschaltung des Ausganges bei Kbus Fehler
	xChannelOut := FALSE XOR fbxInvert.xValue;
ELSE	
	// Invertierung des Wertes bei aktiver Invertierung
	xChannelOut := xValue XOR fbxInvert.xValue;
END_IF

// Write value on defined DO 
IF usiSlot > 0 AND WagoSysDynamicIoMapping.DynIoManager.DynKbusIoManager.coModules.uiModuleCount >= usiSlot THEN
	WagoSysDynamicIoMapping.DynIoManager.DynKbusIoManager.coModules.aIModules[usiSlot].SetProcessOutBit(scAdressOfChanel.uiByteNr,scAdressOfChanel.uiBitNR,xChannelOut,oStatus => oStatus);	
	xOK := TRUE;
ELSE
	xOK	:= FALSE;
END_IF

(* TREND *)
metTrendLog();
END_METHOD

METHOD metConfig
VAR_INPUT
END_VAR
fbConfigFile();

fbxSimulation 					(_usiParaNr := 1, itfConfigFb := fbConfigFile);
fbxSimulationLock				(_usiParaNr := 2, itfConfigFb := fbConfigFile);
fbxInvert						(_usiParaNr := 3, itfConfigFb := fbConfigFile);
fbxSimulationValue				(_usiParaNr := 4, itfConfigFb := fbConfigFile);
END_METHOD

PROPERTY proThisRef_DO : REFERENCE TO fbDO
GET
proThisRef_DO REF= THIS^;
END_GET
END_PROPERTY

PROPERTY P_scfbDO_fbxInvert : CtaSysConfig.ITF_DATATYPE
GET
P_scfbDO_fbxInvert := fbxInvert;
END_GET
END_PROPERTY

PROPERTY P_scfbDO_fbxSimulationValue : CtaSysConfig.ITF_DATATYPE
GET
P_scfbDO_fbxSimulationValue := fbxSimulationValue;
END_GET
END_PROPERTY

PROPERTY P_All_Init : scDO_Para
SET
fbxSimulationLock._WertInit := P_All_Init.xSimulationLock;
fbxInvert._WertInit 		:= P_All_Init.xInvert;
END_SET
END_PROPERTY

METHOD metTrendLog
IF NOT fbTrendLogxValue.ENABLE THEN
	fbTrendLogxValue.ENABLE := TRUE;
	fbTrendLogxValue.KEY	 := CONCAT('SLOT_',CONCAT(TO_STRING(usiSlot),CONCAT('_DO_',TO_STRING(uiChanel))));
END_IF;
fbTrendLogxValue.SET_VALUE	 := xChannelOut;
END_METHOD

PROPERTY proLogName : STRING(100)
GET
proLogName := CONCAT('SLOT_',CONCAT(TO_STRING(usiSlot),CONCAT('_DO_',TO_STRING(uiChanel))));
END_GET
END_PROPERTY

PROPERTY proIsBOOL_IO : BOOL
GET
proIsBOOL_IO := TRUE;
END_GET
END_PROPERTY

END_FUNCTION_BLOCK

// 21 Interface/Visu/ITF_IO_Manager_Visu
INTERFACE ITF_IO_Manager_Visu EXTENDS __SYSTEM.IQueryInterface

PROPERTY proErrNotEnoughIOs : BOOL
GET
END_GET
END_PROPERTY

PROPERTY proNeededMemSize : UDINT
GET
END_GET
END_PROPERTY

PROPERTY proIoInitDone : BOOL
GET
END_GET
END_PROPERTY

PROPERTY proKbusErrSW : BOOL
GET
END_GET
END_PROPERTY

PROPERTY proKbusErrHW : BOOL
GET
END_GET
END_PROPERTY

PROPERTY proMaxIO : INT
GET
END_GET
END_PROPERTY

PROPERTY proAyIOs : ARRAY [1..Parameter.MAX_NUM_OF_IOS] OF ITF_IO
GET
END_GET
END_PROPERTY

PROPERTY proSimOn : BOOL
SET
END_SET
GET
END_GET
END_PROPERTY


PROPERTY proAllowSim : BOOL
GET
END_GET
END_PROPERTY

END_INTERFACE

// 30 Program Organization Units/fb/fbIO_Manager_Alt
{attribute 'linkalways'}
FUNCTION_BLOCK fbIO_Manager_Alt EXTENDS CtaAppBmk.fbBMK IMPLEMENTS ITF_IO_Manager_Visu
VAR_INPUT
END_VAR
VAR_OUTPUT
    xError  :   BOOL;
    xHand   :   BOOL;
END_VAR
VAR	
// Kbus error	
	xKbusError	AT%IX0.0	: BOOL;	
	xKbusWasError			: BOOL;
// Config Missmatch
	uiCountConfigMissmatch	: UINT;
	xConfigMissmatchError	: BOOL;	
// Init
	xIoInitializationDone	: BOOL;
	xCycleStartDelayDone	: BOOL;
	xProcessImgIsUpdated	: BOOL;

// Resource calculations
	uiMemorySize			: UDINT;
	
	iMaxCountedIOs			: INT;
	xErrorNotEnoughIOs		: BOOL;	

// IO Array
	ayIO 					: ARRAY [1..Parameter.MAX_NUM_OF_IOS] OF ITF_IO; // Array containing informations of every single channel
	
// IO Type Arrays
	ayDI 					: ARRAY [1..Parameter.MAX_NUM_OF_DI] OF fbDI;	// Array containing information of every channel of type DI
	ayDO					: ARRAY [1..Parameter.MAX_NUM_OF_DO] OF fbDO;	// Array containing information of every channel of type DO
	ayAI 					: ARRAY [1..Parameter.MAX_NUM_OF_AI] OF fbAI;	// Array containing information of every channel of type AI
	ayAO					: ARRAY [1..Parameter.MAX_NUM_OF_AO] OF fbAO;	// Array containing information of every channel of type AO

// Bus Array Modbus
	ayComTypes				: ARRAY [1..Parameter.MAX_NUM_OF_COMTYPES] OF WagoTypesCom.I_WagoSysComBase; // Array containing information of type WagoTypesCom
	
// IO Counters
	uiNextIO				: UINT := 1;
	
// IO Type Counters
	uiNextDI				: UINT := 1; 	// Index for next DI Module
	uiNextDO				: UINT := 1;	// Index for next DO Module
	uiNextAI				: UINT := 1;	// Index for next AI Module
	uiNextAO 				: UINT := 1;	// Index for next AO Module
	uiNextCOM               : UINT := 1;    // Index for next COM Module
	uiCountDI				: UINT;			// Total amount of DI Modules	
	uiCountDO				: UINT;       	// Total amount of DO Modules	
	uiCountAI				: UINT;       	// Total amount of AI Modules	
	uiCountAO				: UINT;	    	// Total amount of AO Modules
	uiCountCOM              : UINT;         // Total amount of COM Moduls
// Loop counters
	uiModule				: UINT;			// Amount of modules
	uiChannel				: UINT;			// Amount of channels for each module
	
	diForCyclic				: DINT;
	
	diSizeOf				: DINT;	
	
    diCountHand             : DINT;
    fbReportHand            : CtaAppReport.fbReporter;
    fbReportKBusError       : CtaAppReport.fbReporter;  
	fbReportConfigMissmatch	: CtaAppReport.fbReporter;
END_VAR

(* Reset Config Missmatch *)
uiCountConfigMissmatch := 0;
IF NOT xKbusError THEN
	WagoSysDynamicIoMapping.DynIoManager.DynKbusIoManager.updateProcessImages();
	xProcessImgIsUpdated := TRUE;
	
	IF NOT xIoInitializationDone AND_THEN NOT xKbusWasError THEN
	    // Get the total needed memory size for the found valid modules
        uiMemorySize := WagoSysDynamicIoMapping.DynKbusIoManager.udiTotalMemSize;
		// Set the counter variables
		iMaxCountedIOs := 0;
		// IOs common
		uiNextIO:= 1;
		// DI
		uiNextDI:= 1;
		uiCountDI:=0;
		// DO
		uiNextDO:= 1;
		uiCountDO:=0;
		// AI
		uiNextAI:= 1;
		uiCountAI:=0;
		// AO
		uiNextAO:= 1;
		uiCountAO:=0;	
				
		// Check if DynKbusIoManager is initialized and not in error state
		IF WagoSysDynamicIoMapping.DynIoManager.DynKbusIoManager.xIsInit AND NOT WagoSysDynamicIoMapping.DynIoManager.DynKbusIoManager.xIsError	THEN
			
			// Get the overall amount of chanels over all found and valid modules
			FOR uiModule := 1 TO WagoSysDynamicIoMapping.DynIoManager.DynKbusIoManager.coModules.uiModuleCount BY 1 DO
			    IF WagoSysDynamicIoMapping.DynIoManager.DynKbusIoManager.coModules.aIModules[uiModule].eType <> WagoSysDynamicIoMapping.WagoTypesBusServices.eTerminalType.COMPLEX_INOUT THEN 
				    iMaxCountedIOs := iMaxCountedIOs + TO_INT(WagoSysDynamicIoMapping.DynIoManager.DynKbusIoManager.coModules.aIModules[uiModule].uiChannels);
			    END_IF;
			END_FOR	
			
			// Check if there are enough IO's configured in the GlobalConstants gvl
			IF iMaxCountedIOs > Parameter.MAX_NUM_OF_IOS THEN
		
				// ERROR, not enough IOs
				xErrorNotEnoughIOs := TRUE;
	
			ELSE
				
				// Loop through the modules for the amount of found modules
				FOR uiModule := 1 TO WagoSysDynamicIoMapping.DynIoManager.DynKbusIoManager.coModules.uiModuleCount BY 1 DO
			
					// Check if the found module is of type DIGITAL_INPUT
					IF  WagoSysDynamicIoMapping.DynIoManager.DynKbusIoManager.coModules.aIModules[uiModule].eType = WagoSysDynamicIoMapping.WagoTypesBusServices.eTerminalType.DIGITAL_INPUT THEN
						
						// Loop through the channels for the amount of channels the module has
						FOR uiChannel := 1 TO WagoSysDynamicIoMapping.DynIoManager.DynKbusIoManager.coModules.aIModules[uiModule].uiChannels BY 1 DO
							
							// Reference the interfaces
							IF __QUERYINTERFACE(ayDI[uiNextDI],ayIO[uiNextIO]) THEN	
					
								uiCountDI := uiCountDI + 1;	
								
								// Write data on corresponding array index
								ayDI[uiNextDI].proSlot := WagoSysDynamicIoMapping.DynIoManager.DynKbusIoManager.coModules.aIModules[uiModule].usiSlotNumber;
								ayDI[uiNextDI].proChannel := uiChannel;
								ayDI[uiNextDI].proModuleType := enModuleType.Digital_IN;
								ayDI[uiNextDI].proChannelAdress := fcSlotAdress(ayDI[uiNextDI].proSlot,ayDI[uiNextDI].proModuleType,ayDI[uiNextDI].proChannel);
								
								// Count variables up
								uiNextDI := uiNextDI + 1;
								uiNextIO := uiNextIO + 1;						 			
					
							END_IF			
						END_FOR
			
					// Check if the found module is of type DIGITAL_OUTPUT
					ELSIF WagoSysDynamicIoMapping.DynIoManager.DynKbusIoManager.coModules.aIModules[uiModule].eType = WagoSysDynamicIoMapping.WagoTypesBusServices.eTerminalType.DIGITAL_OUTPUT THEN
						
						// Loop through the channels for the amount of channels the module has
						FOR uiChannel := 1 TO WagoSysDynamicIoMapping.DynIoManager.DynKbusIoManager.coModules.aIModules[uiModule].uiChannels BY 1 DO
							
							// Reference the interfaces
							IF __QUERYINTERFACE(ayDO[uiNextDO],ayIO[uiNextIO]) THEN	

								uiCountDO := uiCountDO + 1;				
								
								// Write data on corresponding array index		
								ayDO[uiNextDO].proSlot := WagoSysDynamicIoMapping.DynIoManager.DynKbusIoManager.coModules.aIModules[uiModule].usiSlotNumber;
								ayDO[uiNextDO].proChannel := uiChannel;
								ayDO[uiNextDO].proModuleType := enModuleType.Digital_OUT;
								ayDO[uiNextDO].proChannelAdress := fcSlotAdress(ayDO[uiNextDO].proSlot,ayDO[uiNextDO].proModuleType,ayDO[uiNextDO].proChannel);					
								
								// Count variables up
								uiNextDO := uiNextDO + 1;
								uiNextIO := uiNextIO + 1;
									
							END_IF			
						END_FOR
			
					// Check if the found module is of type COMPLEX_INPUT
					ELSIF WagoSysDynamicIoMapping.DynIoManager.DynKbusIoManager.coModules.aIModules[uiModule].eType = WagoSysDynamicIoMapping.WagoTypesBusServices.eTerminalType.COMPLEX_INPUT THEN
						
						// Loop through the channels for the amount of channels the module has
						FOR uiChannel := 1 TO WagoSysDynamicIoMapping.DynIoManager.DynKbusIoManager.coModules.aIModules[uiModule].uiChannels BY 1 DO
							
							// Reference the interfaces
							IF __QUERYINTERFACE(ayAI[uiNextAI],ayIO[uiNextIO]) THEN	

								uiCountAI := uiCountAI + 1;					
					
								// Write data on corresponding array index
								ayAI[uiNextAI].proSlot := WagoSysDynamicIoMapping.DynIoManager.DynKbusIoManager.coModules.aIModules[uiModule].usiSlotNumber;
								ayAI[uiNextAI].proChannel := uiChannel;
								ayAI[uiNextAI].proModuleType := fcModuleType(WagoSysDynamicIoMapping.DynIoManager.DynKbusIoManager.coModules.aIModules[uiModule].aOrderNumber);
								ayAI[uiNextAI].proChannelAdress := fcSlotAdress(ayAI[uiNextAI].proSlot,ayAI[uiNextAI].proModuleType,ayAI[uiNextAI].proChannel);
								ayAI[uiNextAI].proAyPos := 
								// Count variables up
								uiNextAI := uiNextAI + 1;
								uiNextIO := uiNextIO + 1;																
					
							END_IF			
						END_FOR
			
					// Check if the found module is of type COMPLEX_OUTPUT
					ELSIF WagoSysDynamicIoMapping.DynIoManager.DynKbusIoManager.coModules.aIModules[uiModule].eType = WagoSysDynamicIoMapping.WagoTypesBusServices.eTerminalType.COMPLEX_OUTPUT THEN
			
						// Loop through the channels for the amount of channels the module has
						FOR uiChannel := 1 TO WagoSysDynamicIoMapping.DynIoManager.DynKbusIoManager.coModules.aIModules[uiModule].uiChannels BY 1 DO
							
							// Reference the interfaces
							IF __QUERYINTERFACE(ayAO[uiNextAO],ayIO[uiNextIO]) THEN	
					
								uiCountAO := uiCountAO + 1;
								
								// Write data on corresponding array index
								ayAO[uiNextAO].proSlot := WagoSysDynamicIoMapping.DynIoManager.DynKbusIoManager.coModules.aIModules[uiModule].usiSlotNumber;
								ayAO[uiNextAO].proChannel := uiChannel;
								ayAO[uiNextAO].proModuleType := fcModuleType(WagoSysDynamicIoMapping.DynIoManager.DynKbusIoManager.coModules.aIModules[uiModule].aOrderNumber);
								ayAO[uiNextAO].proChannelAdress := fcSlotAdress(ayAO[uiNextAO].proSlot,ayAO[uiNextAO].proModuleType,ayAO[uiNextAO].proChannel);	

								// Count variables up
								uiNextAO := uiNextAO + 1;
								uiNextIO := uiNextIO + 1;				
					
							END_IF			
						END_FOR					
					
					// Check if the found module is of type COMPLEX_INOUT
					ELSIF WagoSysDynamicIoMapping.DynIoManager.DynKbusIoManager.coModules.aIModules[uiModule].eType = WagoSysDynamicIoMapping.WagoTypesBusServices.eTerminalType.COMPLEX_INOUT THEN
						uiCountCOM := uiCountCOM + 1;
                        // Write data on corresponding array index
                        ayComTypes[uiNextCOM] := WagoSysDynamicIoMapping.DynIoManager.DynKbusIoManager.coModules.aIModules[uiModule].IPorts.I_WagoSysComBase;
                        uiNextCOM := uiNextCOM + 1;
					END_IF;
					fcGetModulImage(TO_USINT(uiModule));
				END_FOR;	
				
				xErrorNotEnoughIOs := FALSE;	
				xIoInitializationDone := TRUE;
			END_IF;			
		END_IF;		
	END_IF;	
ELSE
	// Error: Kbus is in Error state			
	xProcessImgIsUpdated 	:= FALSE;
	xKbusWasError 			:= TRUE;	
END_IF

(* Zyklische aktualisierung *)
IF xIoInitializationDone AND xCycleStartDelayDone THEN	
    diCountHand := 0;
	FOR diForCyclic := LOWER_BOUND(ayIO,1) TO TO_DINT(iMaxCountedIOs) BY 1 DO		
        IF ayIO[diForCyclic] <> 0 THEN
            ayIO[diForCyclic].metCyclicKbus();
            ayIO[diForCyclic].proKbusOk := NOT xKbusError AND NOT xKbusWasError;
            IF ayIO[diForCyclic].proIsHand THEN
                diCountHand := diCountHand + 1;
			END_IF;
        END_IF;
	END_FOR;	
END_IF;
(* Cycle Delay Done *)
xCycleStartDelayDone := TRUE;
(* Report Hand *)
xHand := diCountHand <> 0;
fbReportHand.proHandLokal := xHand;
fbReportHand.proPrio      := 1;
fbReportHand.metReport( xSetReportIn                := xHand,
                        iReportID                   := 91,
                        enReportTypeIn              := CtaAppReport.enReportType.Warning,
                        enReportAcknowledgeTypeIn   := CtaAppReport.enReportacknowledgeType.Auto,
                        tDelay                      := T#0S,
                        ITF_BMK_IN                  := THIS^,
                        pstReportTextListIn         := ADR(GlobalKonstant.stWarningTextList),
                        stOptionalReportText        := '',
                        iRetryTilReportLock         := 0,
                        xResetCount                 := FALSE,
                        tReset                      := T#0S);
(* Report Error *)
fbReportConfigMissmatch.proPrio   := 1;
fbReportConfigMissmatch.metReport(	xSetReportIn                := xConfigMissmatchError,
									iReportID                   := 92,
									enReportTypeIn              := CtaAppReport.enReportType.Error,
									enReportAcknowledgeTypeIn   := CtaAppReport.enReportacknowledgeType.Auto,
									tDelay                      := T#1S,
									ITF_BMK_IN                  := THIS^,
									pstReportTextListIn         := ADR(GlobalKonstant.stErrorTextList),
									stOptionalReportText        := '',
									iRetryTilReportLock         := 0,
									xResetCount                 := FALSE,
									tReset                      := T#0S);

(* Report Error *)
fbReportKBusError.proPrio   := 1;
fbReportKBusError.metReport(		xSetReportIn                := xKbusError OR xKbusWasError,
									iReportID                   := 91,
									enReportTypeIn              := CtaAppReport.enReportType.Error,
									enReportAcknowledgeTypeIn   := CtaAppReport.enReportacknowledgeType.Auto,
									tDelay                      := T#1S,
									ITF_BMK_IN                  := THIS^,
									pstReportTextListIn         := ADR(GlobalKonstant.stErrorTextList),
									stOptionalReportText        := '',
									iRetryTilReportLock         := 0,
									xResetCount                 := FALSE,
									tReset                      := T#0S);
(* Error *)							
xError	:= xKbusError OR xKbusWasError OR xConfigMissmatchError; 
xConfigMissmatchError  := FALSE;

PROPERTY proCycleStartDelayDone : BOOL
GET
END_GET
END_PROPERTY

METHOD metRequestIO_ITF : ITF_IO
VAR_INPUT
	usiSlot 	:	USINT;
	uiChanel	:	UINT;
END_VAR

VAR 
	iIOCounter	: DINT;
END_VAR
(*Count true array of IOs for the amount of IOs in the array*)
FOR iIOCounter := LOWER_BOUND(ayIO,1) TO UPPER_BOUND(ayIO,1) BY 1 DO
	
	IF ayIO[iIOCounter] <> 0 THEN
		(*Search true array until condition matches*)
		IF ayIO[iIOCounter].proSlot = usiSlot AND ayIO[iIOCounter].proChannel = uiChanel THEN
		
			(*Return found interface*)
			metRequestIO_ITF := ayIO[iIOCounter];
			EXIT;	
		END_IF		
	END_IF
END_FOR
END_METHOD

PROPERTY proAyIOs : ARRAY [1..Parameter.MAX_NUM_OF_IOS] OF ITF_IO
GET
proAyIOs := ayIO;
END_GET
END_PROPERTY

PROPERTY proMaxIO : INT
GET
proMaxIO := iMaxCountedIOs;
END_GET
END_PROPERTY

PROPERTY proErrNotEnoughIOs : BOOL
GET
proErrNotEnoughIOs := xErrorNotEnoughIOs;
END_GET
END_PROPERTY

PROPERTY proIoInitDone : BOOL
GET
proIoInitDone := xIoInitializationDone;
END_GET
END_PROPERTY

PROPERTY proKbusErrHW : BOOL
GET
proKbusErrHW := xKbusError;
END_GET
END_PROPERTY

PROPERTY proKbusErrSW : BOOL
GET
proKbusErrSW := xKbusWasError;
END_GET
END_PROPERTY

PROPERTY proNeededMemSize : UDINT
GET
proNeededMemSize := uiMemorySize;
END_GET
END_PROPERTY

METHOD metRequestCOM_ITF : WagoTypesCom.I_WagoSysComBase
VAR_INPUT
	usiSlot 	:	USINT;
END_VAR
IF WagoSysDynamicIoMapping.DynIoManager.DynKbusIoManager.xIsInit AND NOT WagoSysDynamicIoMapping.DynIoManager.DynKbusIoManager.xIsError THEN
	IF usiSlot > 0 AND usiSlot <= WagoSysDynamicIoMapping.DynIoManager.DynKbusIoManager.coModules.uiModuleCount THEN
		IF WagoSysDynamicIoMapping.DynIoManager.DynKbusIoManager.coModules.aIModules[usiSlot].eType = WagoSysDynamicIoMapping.WagoTypesBusServices.eTerminalType.COMPLEX_INOUT THEN
			metRequestCOM_ITF := WagoSysDynamicIoMapping.DynIoManager.DynKbusIoManager.coModules.aIModules[usiSlot].IPorts.I_WagoSysComBase;
		END_IF;
	END_IF;
END_IF;
END_METHOD

METHOD metModulConfigCheck : BOOL
VAR_INPUT
    usiSlot     :   USINT;
	uiOrderNr1	:	UINT;			// Bsp.750
	uiOrderNr2	:	UINT;			// Bsp.455
END_VAR
VAR
    uiModule    :   UINT;
    ayOrderNr   :   ARRAY[0..3] OF UINT;
END_VAR
metModulConfigCheck := FALSE;
IF usiSlot >= 1 AND usiSlot <= 125 THEN
	IF WagoSysDynamicIoMapping.DynIoManager.DynKbusIoManager.xIsInit AND NOT WagoSysDynamicIoMapping.DynIoManager.DynKbusIoManager.xIsError THEN
		uiModule := WagoSysDynamicIoMapping.DynIoManager.DynKbusIoManager.coModules.uiModuleCount;
		IF usiSlot <=  uiModule THEN
			ayOrderNr := WagoSysDynamicIoMapping.DynIoManager.DynKbusIoManager.coModules.aIModules[usiSlot].aOrderNumber;   
			IF ayOrderNr[0] = 750 THEN
				IF fcCheckModul(uiOrderNr1,ayOrderNr[0],uiOrderNr2,ayOrderNr[1]) THEN  
					metModulConfigCheck := TRUE;
				ELSE
					uiCountConfigMissmatch := uiCountConfigMissmatch + 1;
				END_IF;
			(* Lösung da Digital nicht ay Ordernr unterstützt *)
			ELSIF WagoSysDynamicIoMapping.DynIoManager.DynKbusIoManager.coModules.aIModules[usiSlot].eType = WagoTypesBusServices.eTerminalType.DIGITAL_INPUT THEN
				IF WagoSysDynamicIoMapping.DynIoManager.DynKbusIoManager.coModules.aIModules[usiSlot].uiChannels = 16 THEN
					(* 750-1405 *)
					IF fcCheckModul(uiOrderNr1,750,uiOrderNr2,1405) THEN  
						metModulConfigCheck := TRUE;
					ELSE
						uiCountConfigMissmatch := uiCountConfigMissmatch + 1;
					END_IF;     
				ELSIF WagoSysDynamicIoMapping.DynIoManager.DynKbusIoManager.coModules.aIModules[usiSlot].uiChannels = 8 THEN
					(* 750-1415 *)
					IF fcCheckModul(uiOrderNr1,750,uiOrderNr2,1415) THEN  
						metModulConfigCheck := TRUE;
					ELSE
						uiCountConfigMissmatch := uiCountConfigMissmatch + 1;
					END_IF;  
				ELSIF WagoSysDynamicIoMapping.DynIoManager.DynKbusIoManager.coModules.aIModules[usiSlot].uiChannels = 4 THEN
					(* 750-432 *)
					IF fcCheckModul(uiOrderNr1,750,uiOrderNr2,432) THEN  
						metModulConfigCheck := TRUE;
					ELSE
						uiCountConfigMissmatch := uiCountConfigMissmatch + 1;
					END_IF;       
				ELSIF WagoSysDynamicIoMapping.DynIoManager.DynKbusIoManager.coModules.aIModules[usiSlot].uiChannels = 2 THEN
					(* 750-400 *)
					IF fcCheckModul(uiOrderNr1,750,uiOrderNr2,400) THEN  
						metModulConfigCheck := TRUE;
					ELSE
						uiCountConfigMissmatch := uiCountConfigMissmatch + 1;
					END_IF;  
				ELSE
					uiCountConfigMissmatch := uiCountConfigMissmatch + 1;                                        
				END_IF;				
			END_IF;
		ELSE
			uiCountConfigMissmatch := uiCountConfigMissmatch + 1;
		END_IF;	
    END_IF;   
END_IF;
IF uiCountConfigMissmatch > 0 THEN
	xConfigMissmatchError := TRUE;
END_IF;
END_METHOD

END_FUNCTION_BLOCK

// 30 Program Organization Units/IO
PROGRAM IO
VAR
END_VAR

GVL_IO.fbIO_Manager(stObjId := Parameter.SPS_BMK_ID);

END_PROGRAM

// 30 Program Organization Units/fb/fbIO_Manager
{attribute 'linkalways'}
FUNCTION_BLOCK fbIO_Manager EXTENDS CtaAppBmk.fbBMK IMPLEMENTS ITF_IO_Manager_Visu
VAR_INPUT
END_VAR
VAR_OUTPUT
    xError  :   BOOL;
    xHand   :   BOOL;
END_VAR
VAR	
// Kbus error	
	xKbusError	AT%IX0.0	: BOOL;	
	xKbusWasError			: BOOL;
// Config Missmatch
	uiCountConfigMissmatch	: UINT;
	xConfigMissmatchError	: BOOL;	
// Init
	xIoInitializationDone	: BOOL;
	xCycleStartDelayDone	: BOOL;
	xProcessImgIsUpdated	: BOOL;

// Resource calculations
	uiMemorySize			: UDINT;
	
	iMaxCountedIOs			: INT;
	xErrorNotEnoughIOs		: BOOL;	

// IO Array
	ayIO 					: ARRAY [1..Parameter.MAX_NUM_OF_IOS] OF ITF_IO; // Array containing informations of every single channel
	
// IO Type Arrays
	ayDI 					: ARRAY [1..Parameter.MAX_NUM_OF_DI] OF fbDI;	// Array containing information of every channel of type DI
	ayDO					: ARRAY [1..Parameter.MAX_NUM_OF_DO] OF fbDO;	// Array containing information of every channel of type DO
	ayAI 					: ARRAY [1..Parameter.MAX_NUM_OF_AI] OF fbAI;	// Array containing information of every channel of type AI
	ayAO					: ARRAY [1..Parameter.MAX_NUM_OF_AO] OF fbAO;	// Array containing information of every channel of type AO

// Bus Array Modbus
	ayComTypes				: ARRAY [1..Parameter.MAX_NUM_OF_COMTYPES] OF WagoTypesCom.I_WagoSysComBase; // Array containing information of type WagoTypesCom
	
// IO Counters
	uiNextIO				: UINT := 1;
	
// IO Type Counters
	uiNextDI				: UINT := 1; 	// Index for next DI Module
	uiNextDO				: UINT := 1;	// Index for next DO Module
	uiNextAI				: UINT := 1;	// Index for next AI Module
	uiNextAO 				: UINT := 1;	// Index for next AO Module
	uiNextCOM               : UINT := 1;    // Index for next COM Module
	uiCountDI				: UINT;			// Total amount of DI Modules	
	uiCountDO				: UINT;       	// Total amount of DO Modules	
	uiCountAI				: UINT;       	// Total amount of AI Modules	
	uiCountAO				: UINT;	    	// Total amount of AO Modules
	uiCountCOM              : UINT;         // Total amount of COM Moduls
// Simulation
	xSimIsPossible			: BOOL;	
	xSimOn					: BOOL;
	usiBigSimSlot			: UsINT;
// Loop counters
	uiModule				: UINT;			// Amount of modules
	uiChannel				: UINT;			// Amount of channels for each module
	
	diForCyclic				: DINT;
	
	diSizeOf				: DINT;	
	
    diCountHand             : DINT;
    fbReportHand            : CtaAppReport.fbReporter;
    fbReportKBusError       : CtaAppReport.fbReporter;  
	fbReportConfigMissmatch	: CtaAppReport.fbReporter;
END_VAR

(* Reset Config Missmatch *)
uiCountConfigMissmatch := 0;
(* Cycle Delay Done *)
IF xIoInitializationDone THEN
	xCycleStartDelayDone := TRUE;
END_IF;
IF NOT xKbusError THEN
	WagoSysDynamicIoMapping.DynIoManager.DynKbusIoManager.updateProcessImages();
	xProcessImgIsUpdated := TRUE;
	
	IF NOT xIoInitializationDone AND_THEN NOT xKbusWasError THEN
	    // Get the total needed memory size for the found valid modules
        uiMemorySize := WagoSysDynamicIoMapping.DynKbusIoManager.udiTotalMemSize;
		// Set the counter variables
		iMaxCountedIOs := 0;
		// IOs common
		uiNextIO:= 1;
		// DI
		uiNextDI:= 1;
		uiCountDI:=0;
		// DO
		uiNextDO:= 1;
		uiCountDO:=0;
		// AI
		uiNextAI:= 1;
		uiCountAI:=0;
		// AO
		uiNextAO:= 1;
		uiCountAO:=0;	
				
		// Check if DynKbusIoManager is initialized and not in error state
		IF WagoSysDynamicIoMapping.DynIoManager.DynKbusIoManager.xIsInit AND NOT WagoSysDynamicIoMapping.DynIoManager.DynKbusIoManager.xIsError	THEN
			
			// Get the overall amount of chanels over all found and valid modules
			FOR uiModule := 1 TO WagoSysDynamicIoMapping.DynIoManager.DynKbusIoManager.coModules.uiModuleCount BY 1 DO
			    IF WagoSysDynamicIoMapping.DynIoManager.DynKbusIoManager.coModules.aIModules[uiModule].eType <> WagoSysDynamicIoMapping.WagoTypesBusServices.eTerminalType.COMPLEX_INOUT THEN 
				    iMaxCountedIOs := iMaxCountedIOs + TO_INT(WagoSysDynamicIoMapping.DynIoManager.DynKbusIoManager.coModules.aIModules[uiModule].uiChannels);
			    END_IF;
			END_FOR	
			
			// Check if there are enough IO's configured in the GlobalConstants gvl
			IF iMaxCountedIOs > Parameter.MAX_NUM_OF_IOS THEN
		
				// ERROR, not enough IOs
				xErrorNotEnoughIOs := TRUE;
	
			ELSE
				
				// Loop through the modules for the amount of found modules
				FOR uiModule := 1 TO WagoSysDynamicIoMapping.DynIoManager.DynKbusIoManager.coModules.uiModuleCount BY 1 DO
			
					// Check if the found module is of type DIGITAL_INPUT
					IF  WagoSysDynamicIoMapping.DynIoManager.DynKbusIoManager.coModules.aIModules[uiModule].eType = WagoSysDynamicIoMapping.WagoTypesBusServices.eTerminalType.DIGITAL_INPUT THEN
						
						// Loop through the channels for the amount of channels the module has
						FOR uiChannel := 1 TO WagoSysDynamicIoMapping.DynIoManager.DynKbusIoManager.coModules.aIModules[uiModule].uiChannels BY 1 DO
							
							// Reference the interfaces
							IF __QUERYINTERFACE(ayDI[uiNextDI],ayIO[uiNextIO]) THEN	
					
								uiCountDI := uiCountDI + 1;	
								
								// Write data on corresponding array index
								ayDI[uiNextDI].proSlot := WagoSysDynamicIoMapping.DynIoManager.DynKbusIoManager.coModules.aIModules[uiModule].usiSlotNumber;
								ayDI[uiNextDI].proChannel := uiChannel;
								ayDI[uiNextDI].proModuleType := enModuleType.Digital_IN;
								ayDI[uiNextDI].proChannelAdress := fcSlotAdress(ayDI[uiNextDI].proSlot,ayDI[uiNextDI].proModuleType,ayDI[uiNextDI].proChannel);
								
								// Count variables up
								uiNextDI := uiNextDI + 1;
								uiNextIO := uiNextIO + 1;						 			
					
							END_IF			
						END_FOR
			
					// Check if the found module is of type DIGITAL_OUTPUT
					ELSIF WagoSysDynamicIoMapping.DynIoManager.DynKbusIoManager.coModules.aIModules[uiModule].eType = WagoSysDynamicIoMapping.WagoTypesBusServices.eTerminalType.DIGITAL_OUTPUT THEN
						
						// Loop through the channels for the amount of channels the module has
						FOR uiChannel := 1 TO WagoSysDynamicIoMapping.DynIoManager.DynKbusIoManager.coModules.aIModules[uiModule].uiChannels BY 1 DO
							
							// Reference the interfaces
							IF __QUERYINTERFACE(ayDO[uiNextDO],ayIO[uiNextIO]) THEN	

								uiCountDO := uiCountDO + 1;				
								
								// Write data on corresponding array index		
								ayDO[uiNextDO].proSlot := WagoSysDynamicIoMapping.DynIoManager.DynKbusIoManager.coModules.aIModules[uiModule].usiSlotNumber;
								ayDO[uiNextDO].proChannel := uiChannel;
								ayDO[uiNextDO].proModuleType := enModuleType.Digital_OUT;
								ayDO[uiNextDO].proChannelAdress := fcSlotAdress(ayDO[uiNextDO].proSlot,ayDO[uiNextDO].proModuleType,ayDO[uiNextDO].proChannel);					
								
								// Count variables up
								uiNextDO := uiNextDO + 1;
								uiNextIO := uiNextIO + 1;
									
							END_IF			
						END_FOR
			
					// Check if the found module is of type COMPLEX_INPUT
					ELSIF WagoSysDynamicIoMapping.DynIoManager.DynKbusIoManager.coModules.aIModules[uiModule].eType = WagoSysDynamicIoMapping.WagoTypesBusServices.eTerminalType.COMPLEX_INPUT THEN
						
						// Loop through the channels for the amount of channels the module has
						FOR uiChannel := 1 TO WagoSysDynamicIoMapping.DynIoManager.DynKbusIoManager.coModules.aIModules[uiModule].uiChannels BY 1 DO
							
							// Reference the interfaces
							IF __QUERYINTERFACE(ayAI[uiNextAI],ayIO[uiNextIO]) THEN	

								uiCountAI := uiCountAI + 1;					
					
								// Write data on corresponding array index
								ayAI[uiNextAI].proSlot := WagoSysDynamicIoMapping.DynIoManager.DynKbusIoManager.coModules.aIModules[uiModule].usiSlotNumber;
								ayAI[uiNextAI].proChannel := uiChannel;
								ayAI[uiNextAI].proModuleType := fcModuleType(WagoSysDynamicIoMapping.DynIoManager.DynKbusIoManager.coModules.aIModules[uiModule].aOrderNumber);
								ayAI[uiNextAI].proChannelAdress := fcSlotAdress(ayAI[uiNextAI].proSlot,ayAI[uiNextAI].proModuleType,ayAI[uiNextAI].proChannel);
								ayAI[uiNextAI].proAyPos := 
								// Count variables up
								uiNextAI := uiNextAI + 1;
								uiNextIO := uiNextIO + 1;																
					
							END_IF			
						END_FOR
			
					// Check if the found module is of type COMPLEX_OUTPUT
					ELSIF WagoSysDynamicIoMapping.DynIoManager.DynKbusIoManager.coModules.aIModules[uiModule].eType = WagoSysDynamicIoMapping.WagoTypesBusServices.eTerminalType.COMPLEX_OUTPUT THEN
			
						// Loop through the channels for the amount of channels the module has
						FOR uiChannel := 1 TO WagoSysDynamicIoMapping.DynIoManager.DynKbusIoManager.coModules.aIModules[uiModule].uiChannels BY 1 DO
							
							// Reference the interfaces
							IF __QUERYINTERFACE(ayAO[uiNextAO],ayIO[uiNextIO]) THEN	
					
								uiCountAO := uiCountAO + 1;
								
								// Write data on corresponding array index
								ayAO[uiNextAO].proSlot := WagoSysDynamicIoMapping.DynIoManager.DynKbusIoManager.coModules.aIModules[uiModule].usiSlotNumber;
								ayAO[uiNextAO].proChannel := uiChannel;
								ayAO[uiNextAO].proModuleType := fcModuleType(WagoSysDynamicIoMapping.DynIoManager.DynKbusIoManager.coModules.aIModules[uiModule].aOrderNumber);
								ayAO[uiNextAO].proChannelAdress := fcSlotAdress(ayAO[uiNextAO].proSlot,ayAO[uiNextAO].proModuleType,ayAO[uiNextAO].proChannel);	

								// Count variables up
								uiNextAO := uiNextAO + 1;
								uiNextIO := uiNextIO + 1;				
					
							END_IF			
						END_FOR					
					
					// Check if the found module is of type COMPLEX_INOUT
					ELSIF WagoSysDynamicIoMapping.DynIoManager.DynKbusIoManager.coModules.aIModules[uiModule].eType = WagoSysDynamicIoMapping.WagoTypesBusServices.eTerminalType.COMPLEX_INOUT THEN
						uiCountCOM := uiCountCOM + 1;
                        // Write data on corresponding array index
                        ayComTypes[uiNextCOM] := WagoSysDynamicIoMapping.DynIoManager.DynKbusIoManager.coModules.aIModules[uiModule].IPorts.I_WagoSysComBase;
                        uiNextCOM := uiNextCOM + 1;
					END_IF;
					fcGetModulImage(TO_USINT(uiModule));
				END_FOR;	
				
				xErrorNotEnoughIOs := FALSE;	
				xIoInitializationDone := TRUE;
			END_IF;			
		END_IF;		
	END_IF;	
ELSE
	// Error: Kbus is in Error state			
	xProcessImgIsUpdated 	:= FALSE;
	xKbusWasError 			:= TRUE;
	xSimIsPossible 			:= TRUE;
END_IF
(* Simulation *)
IF xSimIsPossible THEN
	IF xSimOn THEN
		IF NOT xIoInitializationDone THEN
			xCycleStartDelayDone := FALSE;
		END_IF;
		xIoInitializationDone := TRUE;
		iMaxCountedIOs := TO_INT(uiNextIO)-1;
	ELSE
		usiBigSimSlot := 0;
	END_IF;
ELSE
	xSimOn := FALSE;
END_IF
(* Zyklische aktualisierung *)
IF xIoInitializationDone AND xCycleStartDelayDone THEN	
    diCountHand := 0;
	FOR diForCyclic := LOWER_BOUND(ayIO,1) TO TO_DINT(iMaxCountedIOs) BY 1 DO		
        IF ayIO[diForCyclic] <> 0 THEN
            ayIO[diForCyclic].metCyclicKbus();
			ayIO[diForCyclic].proiosim := xSimOn;
           	ayIO[diForCyclic].proKbusOk := NOT xKbusError AND NOT xKbusWasError AND NOT xSimOn;
            IF ayIO[diForCyclic].proIsHand THEN
                diCountHand := diCountHand + 1;
			END_IF;
        END_IF;
	END_FOR;	
END_IF;

(* Report Hand *)
xHand := diCountHand <> 0;
fbReportHand.proHandLokal := xHand;
fbReportHand.proPrio      := 1;
fbReportHand.metReport( xSetReportIn                := xHand,
                        iReportID                   := 91,
                        enReportTypeIn              := CtaAppReport.enReportType.Warning,
                        enReportAcknowledgeTypeIn   := CtaAppReport.enReportacknowledgeType.Auto,
                        tDelay                      := T#0S,
                        ITF_BMK_IN                  := THIS^,
                        pstReportTextListIn         := ADR(GlobalKonstant.stWarningTextList),
                        stOptionalReportText        := '',
                        iRetryTilReportLock         := 0,
                        xResetCount                 := FALSE,
                        tReset                      := T#0S);
(* Report Error *)
fbReportConfigMissmatch.proPrio   := 1;
fbReportConfigMissmatch.metReport(	xSetReportIn                := xConfigMissmatchError,
									iReportID                   := 92,
									enReportTypeIn              := CtaAppReport.enReportType.Error,
									enReportAcknowledgeTypeIn   := CtaAppReport.enReportacknowledgeType.Auto,
									tDelay                      := T#1S,
									ITF_BMK_IN                  := THIS^,
									pstReportTextListIn         := ADR(GlobalKonstant.stErrorTextList),
									stOptionalReportText        := '',
									iRetryTilReportLock         := 0,
									xResetCount                 := FALSE,
									tReset                      := T#0S);

(* Report Error *)
fbReportKBusError.proPrio   := 1;
fbReportKBusError.metReport(		xSetReportIn                := xKbusError OR xKbusWasError,
									iReportID                   := 91,
									enReportTypeIn              := CtaAppReport.enReportType.Error,
									enReportAcknowledgeTypeIn   := CtaAppReport.enReportacknowledgeType.Auto,
									tDelay                      := T#1S,
									ITF_BMK_IN                  := THIS^,
									pstReportTextListIn         := ADR(GlobalKonstant.stErrorTextList),
									stOptionalReportText        := '',
									iRetryTilReportLock         := 0,
									xResetCount                 := FALSE,
									tReset                      := T#0S);
(* Error *)							
xError	:= xKbusError OR xKbusWasError OR xConfigMissmatchError; 
xConfigMissmatchError  := FALSE;

PROPERTY proCycleStartDelayDone : BOOL
GET
proCycleStartDelayDone := xCycleStartDelayDone;
END_GET
END_PROPERTY

METHOD metRequestIO_ITF : ITF_IO
VAR_INPUT
	usiSlot 	:	USINT;
	uiChanel	:	UINT;
END_VAR

VAR 
	iIOCounter	: DINT;
END_VAR
(*Count true array of IOs for the amount of IOs in the array*)
FOR iIOCounter := LOWER_BOUND(ayIO,1) TO UPPER_BOUND(ayIO,1) BY 1 DO
	IF ayIO[iIOCounter] <> 0 THEN
		(*Search true array until condition matches*)
		IF ayIO[iIOCounter].proSlot = usiSlot AND ayIO[iIOCounter].proChannel = uiChanel THEN
		
			(*Return found interface*)
			metRequestIO_ITF := ayIO[iIOCounter];
			EXIT;	
		END_IF		
	END_IF
END_FOR
END_METHOD

PROPERTY proAyIOs : ARRAY [1..Parameter.MAX_NUM_OF_IOS] OF ITF_IO
GET
proAyIOs := ayIO;
END_GET
END_PROPERTY

PROPERTY proMaxIO : INT
GET
proMaxIO := iMaxCountedIOs;
END_GET
END_PROPERTY

PROPERTY proErrNotEnoughIOs : BOOL
GET
proErrNotEnoughIOs := xErrorNotEnoughIOs;
END_GET
END_PROPERTY

PROPERTY proIoInitDone : BOOL
GET
proIoInitDone := xIoInitializationDone;
END_GET
END_PROPERTY

PROPERTY proKbusErrHW : BOOL
GET
proKbusErrHW := xKbusError;
END_GET
END_PROPERTY

PROPERTY proKbusErrSW : BOOL
GET
proKbusErrSW := xKbusWasError;
END_GET
END_PROPERTY

PROPERTY proNeededMemSize : UDINT
GET
proNeededMemSize := uiMemorySize;
END_GET
END_PROPERTY

METHOD metRequestCOM_ITF : WagoTypesCom.I_WagoSysComBase
VAR_INPUT
	usiSlot 	:	USINT;
END_VAR
IF WagoSysDynamicIoMapping.DynIoManager.DynKbusIoManager.xIsInit AND NOT WagoSysDynamicIoMapping.DynIoManager.DynKbusIoManager.xIsError THEN
	IF usiSlot > 0 AND usiSlot <= WagoSysDynamicIoMapping.DynIoManager.DynKbusIoManager.coModules.uiModuleCount THEN
		IF WagoSysDynamicIoMapping.DynIoManager.DynKbusIoManager.coModules.aIModules[usiSlot].eType = WagoSysDynamicIoMapping.WagoTypesBusServices.eTerminalType.COMPLEX_INOUT THEN
			metRequestCOM_ITF := WagoSysDynamicIoMapping.DynIoManager.DynKbusIoManager.coModules.aIModules[usiSlot].IPorts.I_WagoSysComBase;
		END_IF;
	END_IF;
END_IF;
END_METHOD

METHOD metModulConfigCheck : BOOL
VAR_INPUT
    usiSlot     :   USINT;
	uiOrderNr1	:	UINT;			// Bsp.750
	uiOrderNr2	:	UINT;			// Bsp.455
END_VAR
VAR
    uiModule    :   UINT;
    ayOrderNr   :   ARRAY[0..3] OF UINT;
END_VAR
metModulConfigCheck := FALSE;
IF NOT xSimOn THEN
	IF usiSlot >= 1 AND usiSlot <= 125 THEN
		IF WagoSysDynamicIoMapping.DynIoManager.DynKbusIoManager.xIsInit AND NOT WagoSysDynamicIoMapping.DynIoManager.DynKbusIoManager.xIsError THEN
			uiModule := WagoSysDynamicIoMapping.DynIoManager.DynKbusIoManager.coModules.uiModuleCount;
			IF usiSlot <=  uiModule THEN
				ayOrderNr := WagoSysDynamicIoMapping.DynIoManager.DynKbusIoManager.coModules.aIModules[usiSlot].aOrderNumber;   
				IF ayOrderNr[0] = 750 THEN
					IF fcCheckModul(uiOrderNr1,ayOrderNr[0],uiOrderNr2,ayOrderNr[1]) THEN  
						metModulConfigCheck := TRUE;
					ELSE
						uiCountConfigMissmatch := uiCountConfigMissmatch + 1;
					END_IF;
				(* Lösung da Digital nicht ay Ordernr unterstützt *)
				ELSIF WagoSysDynamicIoMapping.DynIoManager.DynKbusIoManager.coModules.aIModules[usiSlot].eType = WagoTypesBusServices.eTerminalType.DIGITAL_INPUT THEN
					IF WagoSysDynamicIoMapping.DynIoManager.DynKbusIoManager.coModules.aIModules[usiSlot].uiChannels = 16 THEN
						(* 750-1405 *)
						IF fcCheckModul(uiOrderNr1,750,uiOrderNr2,1405) THEN  
							metModulConfigCheck := TRUE;
						ELSE
							uiCountConfigMissmatch := uiCountConfigMissmatch + 1;
						END_IF;     
					ELSIF WagoSysDynamicIoMapping.DynIoManager.DynKbusIoManager.coModules.aIModules[usiSlot].uiChannels = 8 THEN
						(* 750-1415 *)
						IF fcCheckModul(uiOrderNr1,750,uiOrderNr2,1415) THEN  
							metModulConfigCheck := TRUE;
						ELSIF fcCheckModul(uiOrderNr1,750,uiOrderNr2,430) THEN
							metModulConfigCheck := TRUE;
						ELSE
							uiCountConfigMissmatch := uiCountConfigMissmatch + 1;
						END_IF;  
					ELSIF WagoSysDynamicIoMapping.DynIoManager.DynKbusIoManager.coModules.aIModules[usiSlot].uiChannels = 4 THEN
						(* 750-432 *)
						IF fcCheckModul(uiOrderNr1,750,uiOrderNr2,432) THEN  
							metModulConfigCheck := TRUE;
						ELSE
							uiCountConfigMissmatch := uiCountConfigMissmatch + 1;
						END_IF;       
					ELSIF WagoSysDynamicIoMapping.DynIoManager.DynKbusIoManager.coModules.aIModules[usiSlot].uiChannels = 2 THEN
						(* 750-400 *)
						IF fcCheckModul(uiOrderNr1,750,uiOrderNr2,400) THEN  
							metModulConfigCheck := TRUE;
						ELSE
							uiCountConfigMissmatch := uiCountConfigMissmatch + 1;
						END_IF;  
					ELSE
						uiCountConfigMissmatch := uiCountConfigMissmatch + 1;                                        
					END_IF;				
				END_IF;
			ELSE
				uiCountConfigMissmatch := uiCountConfigMissmatch + 1;
			END_IF;	
		END_IF;   
	END_IF;
ELSE
	IF usiSlot > usiBigSimSlot THEN
		usiBigSimSlot := usiSlot;
		ayOrderNr[0] := uiOrderNr1;
		ayOrderNr[1] := uiOrderNr2;
		 
		 
		// Loop through the channels for the amount of channels the module has
		FOR uiChannel := 1 TO fcSetModulImageForSimAndGetChanels(usiSlot,ayOrderNr) BY 1 DO	
			IF uiNextIO <= Parameter.MAX_NUM_OF_IOS THEN
				IF fcModuleType(ayOrderNr) = enModuleType.DC_0_10V_IN OR fcModuleType(ayOrderNr) = enModuleType.DC_4_20mA_IN OR fcModuleType(ayOrderNr) = enModuleType.OHM THEN
					// Reference the interfaces
					IF uiNextAI <= Parameter.MAX_NUM_OF_AI AND_THEN __QUERYINTERFACE(ayAI[uiNextAI],ayIO[uiNextIO]) THEN	
	
						uiCountAI := uiCountAI + 1;					
			
						// Write data on corresponding array index
						ayAI[uiNextAI].proSlot := usiSlot;
						ayAI[uiNextAI].proChannel := uiChannel;
						ayAI[uiNextAI].proModuleType := fcModuleType(ayOrderNr);
						ayAI[uiNextAI].proChannelAdress := fcSlotAdress(ayAI[uiNextAI].proSlot,ayAI[uiNextAI].proModuleType,ayAI[uiNextAI].proChannel);
						ayAI[uiNextAI].proAyPos := 
						// Count variables up
						uiNextAI := uiNextAI + 1;
						uiNextIO := uiNextIO + 1;																
			
					END_IF		
				ELSIF uiNextAO <= Parameter.MAX_NUM_OF_AO AND_THEN fcModuleType(ayOrderNr) = enModuleType.DC_0_10V_OUT OR fcModuleType(ayOrderNr) = enModuleType.DC_0_20mA_OUT OR fcModuleType(ayOrderNr) = enModuleType.DC_4_20mA_OUT THEN
					// Reference the interfaces
					IF __QUERYINTERFACE(ayAO[uiNextAO],ayIO[uiNextIO]) THEN	
			
						uiCountAO := uiCountAO + 1;
						
						// Write data on corresponding array index
						ayAO[uiNextAO].proSlot := usiSlot;
						ayAO[uiNextAO].proChannel := uiChannel;
						ayAO[uiNextAO].proModuleType := fcModuleType(ayOrderNr);
						ayAO[uiNextAO].proChannelAdress := fcSlotAdress(ayAO[uiNextAO].proSlot,ayAO[uiNextAO].proModuleType,ayAO[uiNextAO].proChannel);	
		
						// Count variables up
						uiNextAO := uiNextAO + 1;
						uiNextIO := uiNextIO + 1;				
					END_IF	
				ELSIF uiNextDI <= Parameter.MAX_NUM_OF_DI AND_THEN fcModuleType(ayOrderNr) = enModuleType.Digital_IN THEN
					// Reference the interfaces
					IF __QUERYINTERFACE(ayDI[uiNextDI],ayIO[uiNextIO]) THEN	
			
						uiCountDI := uiCountDI + 1;	
						
						// Write data on corresponding array index
						ayDI[uiNextDI].proSlot := usiSlot;
						ayDI[uiNextDI].proChannel := uiChannel;
						ayDI[uiNextDI].proModuleType := enModuleType.Digital_IN;
						ayDI[uiNextDI].proChannelAdress := fcSlotAdress(ayDI[uiNextDI].proSlot,ayDI[uiNextDI].proModuleType,ayDI[uiNextDI].proChannel);
						
						// Count variables up
						uiNextDI := uiNextDI + 1;
						uiNextIO := uiNextIO + 1;						 			
			
					END_IF				
				ELSIF fcModuleType(ayOrderNr) = enModuleType.Digital_OUT THEN
					// Reference the interfaces
					IF uiNextDo <= Parameter.MAX_NUM_OF_Do AND_THEN __QUERYINTERFACE(ayDO[uiNextDO],ayIO[uiNextIO]) THEN	
	
						uiCountDO := uiCountDO + 1;				
						
						// Write data on corresponding array index		
						ayDO[uiNextDO].proSlot := usiSlot;
						ayDO[uiNextDO].proChannel := uiChannel;
						ayDO[uiNextDO].proModuleType := enModuleType.Digital_OUT;
						ayDO[uiNextDO].proChannelAdress := fcSlotAdress(ayDO[uiNextDO].proSlot,ayDO[uiNextDO].proModuleType,ayDO[uiNextDO].proChannel);					
						
						// Count variables up
						uiNextDO := uiNextDO + 1;
						uiNextIO := uiNextIO + 1;
							
					END_IF;					
				END_IF;
			END_IF;
		END_FOR;		
	END_IF;
END_IF;
IF uiCountConfigMissmatch > 0 THEN
	xConfigMissmatchError := TRUE;
END_IF;
END_METHOD

PROPERTY proSimOn : BOOL
SET
xSimOn := proSimOn;
END_SET
GET
proSimOn := xSimOn;
END_GET
END_PROPERTY


PROPERTY proAllowSim : BOOL
GET
proAllowSim := xSimIsPossible;
END_GET
END_PROPERTY

END_FUNCTION_BLOCK

// 30 Program Organization Units/fc/Adresse/fcSlotAdress
(*Funktion zur Definition der Byte und Bit Adresse eines IO Chanels anhand des Modultyps*)
FUNCTION fcSlotAdress : scChanelAdress
VAR_INPUT
	uiSlot			:	UINT;
	enModulType		:	enModuleType;
	uiChannel		: 	UINT;
END_VAR

CASE enModulType OF
	
	// Errechnung der Byte- Bit Nummer eines digitalen Modules 
	enModuleType.Digital_IN,enModuleType.Digital_OUT:
		
		// Definition der Byte- Bit Nummer abhängig der Channel- Nummer
		IF uiChannel - 1 <= 7 THEN	
			fcSlotAdress.uiByteNr := 0;
			fcSlotAdress.uiBitNR := UINT_TO_USINT(uiChannel - 1);
			
		ELSIF uiChannel - 1 >= 8 AND uiChannel - 1 <= 15 THEN
			fcSlotAdress.uiByteNr  := 1;
			fcSlotAdress.uiBitNR := UINT_TO_USINT((uiChannel - 1) - 8);	

		ELSIF uiChannel - 1 >= 16 AND uiChannel - 1 <= 24 THEN
			fcSlotAdress.uiByteNr := 2;
			fcSlotAdress.uiBitNR := UINT_TO_USINT((uiChannel - 1) - 16);
		END_IF
	
	// Errechnung der Byte- Nummer eines Analogen Modules	
	enModuleType.DC_0_10V_IN,enModuleType.DC_0_10V_OUT,
	enModuleType.DC_4_20mA_IN,enModuleType.DC_4_20mA_OUT,
	enModuleType.ohm:
		
		// Definition der Byte- Nummer abhängig der Channel- Nummer
		CASE uiChannel OF
		
			1: // Chanel 1				
				fcSlotAdress.uiByteNr := 0;				
							 
			2: // Chanel 2			
				fcSlotAdress.uiByteNr := 2;
							 
			3: // Chanel 3		
				fcSlotAdress.uiByteNr := 4;
							 
			4: // Chanel 4		
				fcSlotAdress.uiByteNr := 6;
							 
			5: // Chanel 5		
				fcSlotAdress.uiByteNr := 8;

			6: // Chanel 6			
				fcSlotAdress.uiByteNr := 10;
							 
			7: // Chanel 7			
				fcSlotAdress.uiByteNr := 12;
							 
			8: // Chanel 8			
				fcSlotAdress.uiByteNr := 14;
	
		END_CASE
		
		// Definition der Bit- Nummer, bei Analogmodulen standardmässig 0
		fcSlotAdress.uiBitNR := 0;
	
END_CASE

END_FUNCTION

// 30 Program Organization Units/fc/Modul/fcModuleType
(*Funktion zur Definition des Modultyps anhang der Herstellernummer*) 
FUNCTION fcModuleType : enModuleType
VAR_INPUT
	ayOrderNr	: ARRAY [0..3] OF UINT;
END_VAR

IF ayOrderNr[0] = 750 THEN
    // 4-Kanal-Analogeingang 0..10V DC
    IF ayOrderNr[1] = 459 THEN
        
        fcModuleType := enModuleType.DC_0_10V_IN;
    
    // 8-Kanal-Analogausgang 0..10V DC	
    ELSIF ayOrderNr[1] = 597 THEN	
        
        fcModuleType := enModuleType.DC_0_10V_OUT;
    
    // 4-Kanal-Analogeingang 4..20 mA DC ohne DC Versorgung
    ELSIF ayOrderNr[1] = 455 THEN
        
        fcModuleType := enModuleType.DC_4_20mA_IN;
    
    // 2-Kanal-Analogeingang 4..20 mA DC mit DC Versorgung
    ELSIF ayOrderNr[1] = 466 THEN
        
        fcModuleType := enModuleType.DC_4_20mA_IN;
    
    // 8-Kanal-Analogeingang Widerstandsmessung			
    ELSIF ayOrderNr[1] = 451 THEN
        
        fcModuleType := enModuleType.ohm;
		
    // 4-Kanal-Analogausgang 4-20mA			
    ELSIF ayOrderNr[1] = 555 THEN
        
        fcModuleType := enModuleType.DC_4_20mA_OUT;        

    // 4-Kanal-Analogausgang 0-20mA			
    ELSIF ayOrderNr[1] = 553 THEN
        
        fcModuleType := enModuleType.DC_0_20mA_OUT;        		
		
    // RS485		
    ELSIF ayOrderNr[1] = 652 OR ayOrderNr[1] = 653 THEN
        
        fcModuleType := enModuleType.RS485;

    // 4-Kanal-Relais Out 			
    ELSIF ayOrderNr[1] = 515 THEN
        
        fcModuleType := enModuleType.Digital_OUT;
		
     // 16-Kanal-Digital Out 			
    ELSIF ayOrderNr[1] = 1504 THEN
        
        fcModuleType := enModuleType.Digital_OUT; 	

     // 16-Kanal-Digital In 			
    ELSIF ayOrderNr[1] = 1405 THEN
        
        fcModuleType := enModuleType.Digital_IN; 	

     // 8-Kanal-Digital In 			
    ELSIF ayOrderNr[1] = 1415 THEN
        
        fcModuleType := enModuleType.Digital_IN; 	
		
     // 8-Kanal-Digital In 			
    ELSIF ayOrderNr[1] = 430 THEN
        
        fcModuleType := enModuleType.Digital_IN; 
		
     // 4-Kanal-Digital In 			
    ELSIF ayOrderNr[1] = 432 THEN
        
        fcModuleType := enModuleType.Digital_IN; 	
  
     // 2-Kanal-Digital In 			
    ELSIF ayOrderNr[1] = 400 THEN
        
        fcModuleType := enModuleType.Digital_IN; 	
   
    // Modul nicht bekannt
    ELSE
        
        fcModuleType := enModuleType.Unknown;	
        
    END_IF;
ELSE
    fcModuleType := enModuleType.Unknown;	
END_IF;

END_FUNCTION

// 30 Program Organization Units/fc/Terminal Visu/fcGetModulImage
FUNCTION fcGetModulImage : STRING
VAR_INPUT
    usiSlot     :   USINT;
END_VAR
VAR
    uiModule    :   UINT;
    ayOrderNr   :   ARRAY[0..3] OF UINT;
END_VAR

IF usiSlot >= 1 AND usiSlot <= 125 THEN
	IF GVL_IO_TERMINALS.aystIoTerminalType[usiSlot] = '' THEN
		IF WagoSysDynamicIoMapping.DynIoManager.DynKbusIoManager.xIsInit AND NOT WagoSysDynamicIoMapping.DynIoManager.DynKbusIoManager.xIsError THEN
			uiModule := WagoSysDynamicIoMapping.DynIoManager.DynKbusIoManager.coModules.uiModuleCount;
			IF usiSlot <=  uiModule THEN
				ayOrderNr := WagoSysDynamicIoMapping.DynIoManager.DynKbusIoManager.coModules.aIModules[usiSlot].aOrderNumber;   
				IF ayOrderNr[0] = 750 THEN  
					(* 750-451 *)
					IF ayOrderNr[1] = 451 THEN
						fcGetModulImage := 'IO_TERMINALS.0750_451';    
					(* 750-455 *)
					ELSIF ayOrderNr[1] = 455 THEN
						fcGetModulImage := 'IO_TERMINALS.0750_455';   
					(* 750-459 *)
					ELSIF ayOrderNr[1] = 459 THEN
						fcGetModulImage := 'IO_TERMINALS.0750_459';   
					(* 750-466 *)
					ELSIF ayOrderNr[1] = 466 THEN
						fcGetModulImage := 'IO_TERMINALS.0750_466';    
					(* 750-597 *)
					ELSIF ayOrderNr[1] = 555 THEN
						fcGetModulImage := 'IO_TERMINALS.0750_555';   
					(* 750-597 *)
					ELSIF ayOrderNr[1] = 597 THEN
						fcGetModulImage := 'IO_TERMINALS.0750_597';    
					(* 750-652 *)
					ELSIF ayOrderNr[1] = 652 THEN
						fcGetModulImage := 'IO_TERMINALS.0750_652';     
					ELSE
					(* BLANK *)
						fcGetModulImage := 'IO_TERMINALS.0750_BLANK';      
					END_IF;
				(* DI *)
				ELSIF WagoSysDynamicIoMapping.DynIoManager.DynKbusIoManager.coModules.aIModules[usiSlot].eType = WagoTypesBusServices.eTerminalType.DIGITAL_INPUT THEN
					IF WagoSysDynamicIoMapping.DynIoManager.DynKbusIoManager.coModules.aIModules[usiSlot].uiChannels = 16 THEN
						(* 750-1405 *)
						fcGetModulImage := 'IO_TERMINALS.0750_1405';          
					ELSIF WagoSysDynamicIoMapping.DynIoManager.DynKbusIoManager.coModules.aIModules[usiSlot].uiChannels = 8 THEN
						(* 750-1415 *)
						fcGetModulImage := 'IO_TERMINALS.0750_1415';   
					ELSIF WagoSysDynamicIoMapping.DynIoManager.DynKbusIoManager.coModules.aIModules[usiSlot].uiChannels = 4 THEN
						(* 750-432 *)
						fcGetModulImage := 'IO_TERMINALS.0750_432';          
					ELSIF WagoSysDynamicIoMapping.DynIoManager.DynKbusIoManager.coModules.aIModules[usiSlot].uiChannels = 2 THEN
						(* 750-400 *)
						fcGetModulImage := 'IO_TERMINALS.0750_400';  
					ELSE
						(* 750-400 *)
						fcGetModulImage := 'IO_TERMINALS.0750_400';                                          
					END_IF;   
				(* DO *)  
				ELSIF WagoSysDynamicIoMapping.DynIoManager.DynKbusIoManager.coModules.aIModules[usiSlot].eType = WagoTypesBusServices.eTerminalType.DIGITAL_OUTPUT THEN
					IF WagoSysDynamicIoMapping.DynIoManager.DynKbusIoManager.coModules.aIModules[usiSlot].uiChannels = 16 THEN
						(* 750-1504 *)
						fcGetModulImage := 'IO_TERMINALS.0750_1504'; 
					ELSE	
						(* 750-515 *)
						fcGetModulImage := 'IO_TERMINALS.0750_515';   
					END_IF;            
				END_IF;
			ELSIF uiModule + 1 = usiSlot THEN
				(* End Modul *)
				fcGetModulImage := 'IO_TERMINALS.0750_600';
			ELSE 
				(* Empty *)
				fcGetModulImage := '';
			END_IF;
			GVL_IO_TERMINALS.aystIoTerminalType[usiSlot] := fcGetModulImage;
		END_IF;
	ELSE
		fcGetModulImage := GVL_IO_TERMINALS.aystIoTerminalType[usiSlot];		
    END_IF;   
END_IF;

END_FUNCTION

// 30 Program Organization Units/fc/ModulCheck/fcCheckModul
FUNCTION fcCheckModul : BOOL
VAR_INPUT
	uiOrderNr1Usr	:	UINT;			// Bsp.750
	uiOrderNr1Mod	:	UINT;			// Bsp.750
	uiOrderNr2Usr	:	UINT;			// Bsp.455
	uiOrderNr2Mod	:	UINT;			// Bsp.455
END_VAR
VAR
	uiErsatz		:	UINT;
END_VAR

(* Ersatzartikel Prüfen *)
IF uiOrderNr1Usr = 750 AND uiOrderNr2Usr = 466 THEN
	uiErsatz := 455;	
END_IF;

(* Prüfung *)
IF uiOrderNr1Usr = uiOrderNr1Mod AND ( uiOrderNr2Usr = uiOrderNr2Mod OR uiErsatz = uiOrderNr2Mod ) THEN
	fcCheckModul := TRUE;
END_IF;

END_FUNCTION

// 30 Program Organization Units/fc/Terminal Visu/fcSetModulImageForSimAndGetChanels
FUNCTION fcSetModulImageForSimAndGetChanels : UINT
VAR_INPUT
    usiSlot     :   USINT;
	ayOrderNr   :   ARRAY[0..3] OF UINT;
END_VAR

IF usiSlot >= 1 AND usiSlot <= 125 THEN
	IF ayOrderNr[0] = 750 THEN  
		(* 750-451 *)
		IF ayOrderNr[1] = 451 THEN
			GVL_IO_TERMINALS.aystIoTerminalType[usiSlot] := 'IO_TERMINALS.0750_451';
			fcSetModulImageForSimAndGetChanels := 8; 
		(* 750-455 *)
		ELSIF ayOrderNr[1] = 455 THEN
			 GVL_IO_TERMINALS.aystIoTerminalType[usiSlot] := 'IO_TERMINALS.0750_455';  
			 fcSetModulImageForSimAndGetChanels := 4; 
		(* 750-459 *)
		ELSIF ayOrderNr[1] = 459 THEN
			 GVL_IO_TERMINALS.aystIoTerminalType[usiSlot] := 'IO_TERMINALS.0750_459';  
			  fcSetModulImageForSimAndGetChanels := 4;  
		(* 750-466 *)
		ELSIF ayOrderNr[1] = 466 THEN
			 GVL_IO_TERMINALS.aystIoTerminalType[usiSlot] := 'IO_TERMINALS.0750_466'; 
			 fcSetModulImageForSimAndGetChanels := 2;   
		(* 750-555 *)
		ELSIF ayOrderNr[1] = 555 THEN
			 GVL_IO_TERMINALS.aystIoTerminalType[usiSlot] := 'IO_TERMINALS.0750_555'; 
			 fcSetModulImageForSimAndGetChanels := 4;   
		(* 750-597 *)
		ELSIF ayOrderNr[1] = 597 THEN
			 GVL_IO_TERMINALS.aystIoTerminalType[usiSlot] := 'IO_TERMINALS.0750_597';  
			 fcSetModulImageForSimAndGetChanels := 8; 
		(* 750-652 *)
		ELSIF ayOrderNr[1] = 652 THEN
			 GVL_IO_TERMINALS.aystIoTerminalType[usiSlot] := 'IO_TERMINALS.0750_652';    
			 fcSetModulImageForSimAndGetChanels := 0;
		(* 750-1405 *)
		ELSIF ayOrderNr[1] = 1405 THEN
			 GVL_IO_TERMINALS.aystIoTerminalType[usiSlot] := 'IO_TERMINALS.0750_1405';  
			 fcSetModulImageForSimAndGetChanels := 16;
		(* 750-1415 *)
		ELSIF ayOrderNr[1] = 1415 OR ayOrderNr[1] = 0430 THEN
			GVL_IO_TERMINALS.aystIoTerminalType[usiSlot] := 'IO_TERMINALS.0750_1415'; 
			fcSetModulImageForSimAndGetChanels := 8; 	 
		(* 750-432 *)
		ELSIF ayOrderNr[1] = 432 THEN
			 GVL_IO_TERMINALS.aystIoTerminalType[usiSlot] := 'IO_TERMINALS.0750_432';  	
			 fcSetModulImageForSimAndGetChanels := 4;
		(* 750-400 *)
		ELSIF ayOrderNr[1] = 400 THEN
			 GVL_IO_TERMINALS.aystIoTerminalType[usiSlot] := 'IO_TERMINALS.0750_400';  		
			 fcSetModulImageForSimAndGetChanels := 2;
		(* 750-515 *)
		ELSIF ayOrderNr[1] = 515 THEN
			GVL_IO_TERMINALS.aystIoTerminalType[usiSlot] := 'IO_TERMINALS.0750_515';  
 			fcSetModulImageForSimAndGetChanels := 4;
		(* 750-600 *)
		ELSIF ayOrderNr[1] = 600 THEN
			GVL_IO_TERMINALS.aystIoTerminalType[usiSlot] := 'IO_TERMINALS.0750_600'; 
			fcSetModulImageForSimAndGetChanels := 0;	
		(* 750-1504 *)
		ELSIF ayOrderNr[1] = 1504 THEN
			GVL_IO_TERMINALS.aystIoTerminalType[usiSlot] := 'IO_TERMINALS.0750_1504'; 
			fcSetModulImageForSimAndGetChanels := 16;		
		ELSE
			(* BLANK *)
			 GVL_IO_TERMINALS.aystIoTerminalType[usiSlot] := 'IO_TERMINALS.0750_BLANK';   
			fcSetModulImageForSimAndGetChanels := 0;
		END_IF;
		(* 750-600 *)
		IF ayOrderNr[1] <> 600 AND usiSlot < 125 THEN
			GVL_IO_TERMINALS.aystIoTerminalType[usiSlot + 1] := 'IO_TERMINALS.0750_600'; 
		END_IF;		
	END_IF;
END_IF;

END_FUNCTION

// 30 Program Organization Units/fc/ITF_Prüfung/fc_ITF_Evaluation
FUNCTION fc_ITF_Evaluation : ITF_IO
VAR_INPUT
	usiSlot 			:	USINT;
	uiChannel			:	UINT;
END_VAR
VAR
	_ITF_IO				:	ITF_IO;
END_VAR
VAR_OUTPUT
	xEmptyInterface	:	BOOL;
END_VAR

_ITF_IO := GVL_IO.fbIO_Manager.metRequestIO_ITF(usiSlot,uiChannel);

IF	_ITF_IO <> 0 THEN
	fc_ITF_Evaluation := _ITF_IO;
	xEmptyInterface := FALSE;
ELSE
	xEmptyInterface := TRUE;
END_IF

END_FUNCTION

// 30 Program Organization Units/fb/visuhilfe/fbPfcVisuHelp
FUNCTION_BLOCK fbPfcVisuHelp
VAR_OUTPUT
END_VAR
VAR
    usiOldSlot      : USINT;
    iOldZeile       : INT;
    iSlotZeile      : INT;
    ayShowChanel    : ARRAY[1..16] OF BOOL;
    iScrollBar      : INT;
    iOldScrollBar   : INT;
	iFrameSize		: INT;
	rFactor			: REAL := 1;
END_VAR

METHOD metGetSlotIos : INT
VAR_INPUT
    ayIOs			    :	ARRAY [1..Parameter.MAX_NUM_OF_IOS] OF ITF_IO;
    iMax                :   INT;
    iChannel            :   INT;
END_VAR
VAR_IN_OUT
    iZeile              :   INT;
    usiSlot             :   USINT;
END_VAR
VAR
    iFor                :   INT;
END_VAR
(* Zeilen änderung Detektieren *)
IF iZeile <> iOldZeile THEN
    IF iZeile >= 1 AND iZeile <= iMax THEN
        iSlotZeile      := ayIOs[iZeile].proSlot; 
        usiSlot         := TO_USINT(iSlotZeile);
        usiOldSlot      := usiSlot;
        iOldZeile       := iZeile;
        iScrollBar      := metCalcScrollBar(usiSlot);
        iOldScrollBar   := iScrollBar;
    END_IF;    
END_IF;
(* Slot änderung Detektieren *)
IF usiSlot <> usiOldSlot THEN
    FOR iFor := 1 TO TO_INT(iMax) DO
        IF usiSlot = ayIOs[iFor].proSlot THEN
            iSlotZeile      := usiSlot;
            iZeile          := iFor;
            iScrollBar      := metCalcScrollBar(usiSlot);
            iOldScrollBar   := iScrollBar;
            EXIT;    
        END_IF;
    END_FOR;     
    usiOldSlot  := usiSlot;       
END_IF;
(* ScrollBar änderung Detektieren *)
IF iScrollBar <> iOldScrollBar THEN
    usiSlot       := metCalcSlotFromScrollBar(iScrollBar);
    iOldScrollBar := iScrollBar;      
END_IF;
(* IO ITF ausgeben *)
FOR iFor := 1 TO TO_INT(iMax) DO
    IF iSlotZeile = ayIOs[iFor].proSlot THEN
        IF iChannel = ayIOs[iFor].proChannel THEN
            metGetSlotIos := iFor;
            EXIT;    
        END_IF;   
	END_IF;
END_FOR;
(* Check if its Valid Slot *)
IF metGetSlotIos = 0 THEN
    ayShowChanel[LIMIT(1,iChannel,16)] := FALSE;
ELSE
    ayShowChanel[LIMIT(1,iChannel,16)] := TRUE;
END_IF
(* Limit fore Safety array use *)
metGetSlotIos := LIMIT(1,metGetSlotIos,TO_INT(iMax));
END_METHOD

